DECL FDAT FP589={TOOL_NO 0,BASE_NO 0,IPO_FRAME #BASE,POINT2[] " ",TQ_STATE FALSE}
DECL E6POS XP589={X 12666.37592,Y -538.48386,Z 3708.53974,A -127.07895,B -20.60151,C -3.44033,S 2,T 35,E1 -10812.08896,E2 0,E3 0,E4 0,E5 0,E6 0}
; DECL LDAT LCPDATP113={VEL 1,ACC 100,APO_DIST 100,APO_FAC 50.0,ORI_TYP #VAR,CIRC_TYP #BASE,JERK_FAC 50.0}
DECL FDAT FP590={TOOL_NO 0,BASE_NO 0,IPO_FRAME #BASE,POINT2[] " ",TQ_STATE FALSE}
DECL E6POS XP590={X 6379.94734,Y -681.40788,Z 3158.20554,A -102.40256,B 11.37187,C 4.81103,S 2,T 35,E1 -4209.91162,E2 0,E3 0,E4 0,E5 0,E6 0}
; DECL LDAT LCPDATP114={VEL 1,ACC 100,APO_DIST 100,APO_FAC 50.0,ORI_TYP #VAR,CIRC_TYP #BASE,JERK_FAC 50.0}
DECL FDAT FP591={TOOL_NO 0,BASE_NO 0,IPO_FRAME #BASE,POINT2[] " ",TQ_STATE FALSE}
DECL E6POS XP591={X 6328.481,Y -681.40737,Z 3158.20597,A -102.7078,B 7.77597,C 4.76025,S 2,T 35,E1 -4158.44503,E2 0,E3 0,E4 0,E5 0,E6 0}
; DECL LDAT LCPDATP115={VEL 1,ACC 100,APO_DIST 100,APO_FAC 50.0,ORI_TYP #VAR,CIRC_TYP #BASE,JERK_FAC 50.0}
DECL FDAT FP592={TOOL_NO 0,BASE_NO 0,IPO_FRAME #BASE,POINT2[] " ",TQ_STATE FALSE}
DECL E6POS XP592={X 12929.38089,Y -681.40737,Z 3158.20639,A -83.4604,B -12.81532,C -0.94267,S 2,T 35,E1 -10812.08896,E2 0,E3 0,E4 0,E5 0,E6 0}
; DECL LDAT LCPDATP116={VEL 1,ACC 100,APO_DIST 100,APO_FAC 50.0,ORI_TYP #VAR,CIRC_TYP #BASE,JERK_FAC 50.0}
DECL FDAT FP593={TOOL_NO 0,BASE_NO 0,IPO_FRAME #BASE,POINT2[] " ",TQ_STATE FALSE}
DECL E6POS XP593={X 12886.08572,Y -646.4113,Z 3336.02814,A -83.4604,B -12.81532,C -0.94267,S 2,T 35,E1 -10812.08896,E2 0,E3 0,E4 0,E5 0,E6 0}
; DECL LDAT LCPDATP117={VEL 1,ACC 100,APO_DIST 100,APO_FAC 50.0,ORI_TYP #VAR,CIRC_TYP #BASE,JERK_FAC 50.0}
DECL FDAT FP594={TOOL_NO 0,BASE_NO 0,IPO_FRAME #BASE,POINT2[] " ",TQ_STATE FALSE}
DECL E6POS XP594={X 6226.20694,Y -691.76303,Z 3410.82553,A -102.7078,B 7.77597,C 4.76022,S 2,T 35,E1 -4167.06683,E2 0,E3 0,E4 0,E5 0,E6 0}
; DECL LDAT LCPDATP118={VEL 1,ACC 100,APO_DIST 100,APO_FAC 50.0,ORI_TYP #VAR,CIRC_TYP #BASE,JERK_FAC 50.0}
DECL FDAT FP595={TOOL_NO 0,BASE_NO 0,IPO_FRAME #BASE,POINT2[] " ",TQ_STATE FALSE}
DECL E6POS XP595={X 6109.20944,Y -705.3695,Z 3654.40552,A -102.70779,B 7.77597,C 4.76025,S 2,T 35,E1 -4140.9372,E2 0,E3 0,E4 0,E5 0,E6 0}
; DECL LDAT LCPDATP121={VEL 1,ACC 100,APO_DIST 100,APO_FAC 50.0,ORI_TYP #VAR,CIRC_TYP #BASE,JERK_FAC 50.0}
DECL FDAT FP596={TOOL_NO 0,BASE_NO 0,IPO_FRAME #BASE,POINT2[] " ",TQ_STATE FALSE}
DECL E6POS XP596={X 12777.06723,Y -602.17839,Z 3573.69413,A -83.4604,B -12.81532,C -0.94267,S 2,T 35,E1 -10812.08896,E2 0,E3 0,E4 0,E5 0,E6 0}
; DECL LDAT LCPDATP122={VEL 1,ACC 100,APO_DIST 100,APO_FAC 50.0,ORI_TYP #VAR,CIRC_TYP #BASE,JERK_FAC 50.0}
DECL FDAT FP597={TOOL_NO 0,BASE_NO 0,IPO_FRAME #BASE,POINT2[] " ",TQ_STATE FALSE}
DECL E6POS XP597={X 12675.92788,Y -569.18264,Z 3775.2407,A -83.4604,B -12.81532,C -0.94267,S 2,T 35,E1 -10812.08896,E2 0,E3 0,E4 0,E5 0,E6 0}
; DECL LDAT LCPDATP119={VEL 1,ACC 100,APO_DIST 100,APO_FAC 50.0,ORI_TYP #VAR,CIRC_TYP #BASE,JERK_FAC 50.0}
DECL FDAT FP598={TOOL_NO 0,BASE_NO 0,IPO_FRAME #BASE,POINT2[] " ",TQ_STATE FALSE}
DECL E6POS XP598={X 6034.81499,Y -708.12179,Z 3847.76366,A -102.7078,B 7.77596,C 4.76026,S 2,T 35,E1 -4174.36752,E2 0,E3 0,E4 0,E5 0,E6 0}
; DECL LDAT LCPDATP120={VEL 1,ACC 100,APO_DIST 100,APO_FAC 50.0,ORI_TYP #VAR,CIRC_TYP #BASE,JERK_FAC 50.0}
DECL FDAT FP599={TOOL_NO 0,BASE_NO 0,IPO_FRAME #BASE,POINT2[] " ",TQ_STATE FALSE}
DECL E6POS XP599={X 5808.56571,Y -717.10091,Z 4003.7046,A -102.70779,B 7.77596,C 4.76025,S 2,T 35,E1 -4005.10214,E2 0,E3 0,E4 0,E5 0,E6 0}
; DECL LDAT LCPDATP123={VEL 1,ACC 100,APO_DIST 100,APO_FAC 50.0,ORI_TYP #VAR,CIRC_TYP #BASE,JERK_FAC 50.0}
DECL FDAT FP600={TOOL_NO 0,BASE_NO 0,IPO_FRAME #BASE,POINT2[] " ",TQ_STATE FALSE}
DECL E6POS XP600={X 12607.03936,Y -538.48386,Z 3940.5062,A -83.4604,B -12.81532,C -0.94267,S 2,T 35,E1 -10812.08896,E2 0,E3 0,E4 0,E5 0,E6 0}
; DECL LDAT LCPDATP124={VEL 1,ACC 100,APO_DIST 100,APO_FAC 50.0,ORI_TYP #VAR,CIRC_TYP #BASE,JERK_FAC 50.0}
DECL FDAT FP601={TOOL_NO 0,BASE_NO 0,IPO_FRAME #BASE,POINT2[] " ",TQ_STATE FALSE}
DECL E6POS XP601={X 12329.73693,Y -538.48386,Z 3940.5062,A -83.38777,B -15.32829,C -1.2413,S 2,T 35,E1 -10812.08896,E2 0,E3 0,E4 0,E5 0,E6 0}
; DECL LDAT LCPDATP130={VEL 1,ACC 100,APO_DIST 100,APO_FAC 50.0,ORI_TYP #VAR,CIRC_TYP #BASE,JERK_FAC 50.0}
DECL FDAT FP602={TOOL_NO 0,BASE_NO 0,IPO_FRAME #BASE,POINT2[] " ",TQ_STATE FALSE}
DECL E6POS XP602={X 6035.27715,Y -717.10158,Z 4003.70466,A -106.51042,B 6.34838,C 5.00917,S 2,T 35,E1 -4231.81368,E2 0,E3 0,E4 0,E5 0,E6 0}
; DECL LDAT LCPDATP131={VEL 1,ACC 100,APO_DIST 100,APO_FAC 50.0,ORI_TYP #VAR,CIRC_TYP #BASE,JERK_FAC 50.0}
DECL FDAT FP603={TOOL_NO 0,BASE_NO 0,IPO_FRAME #BASE,POINT2[] " ",TQ_STATE FALSE}
DECL E6POS XP603={X 6001.84737,Y -717.10113,Z 4003.70421,A -106.4599,B 4.5615,C 5.54032,S 2,T 35,E1 -4198.38336,E2 0,E3 0,E4 0,E5 0,E6 0}
; DECL LDAT LCPDATP125={VEL 1,ACC 100,APO_DIST 100,APO_FAC 50.0,ORI_TYP #VAR,CIRC_TYP #BASE,JERK_FAC 50.0}
DECL FDAT FP604={TOOL_NO 0,BASE_NO 0,IPO_FRAME #BASE,POINT2[] " ",TQ_STATE FALSE}
DECL E6POS XP604={X 12327.62864,Y -538.48366,Z 3940.50597,A -87.76623,B -17.49847,C -1.50503,S 2,T 35,E1 -10473.34117,E2 0,E3 0,E4 0,E5 0,E6 0}
; DECL LDAT LCPDATP126={VEL 1,ACC 100,APO_DIST 100,APO_FAC 50.0,ORI_TYP #VAR,CIRC_TYP #BASE,JERK_FAC 50.0}
DECL FDAT FP605={TOOL_NO 0,BASE_NO 0,IPO_FRAME #BASE,POINT2[] " ",TQ_STATE FALSE}
DECL E6POS XP605={X 12344.44126,Y -538.48354,Z 3940.50612,A -92.12133,B -19.55447,C -1.59012,S 2,T 35,E1 -10490.15446,E2 0,E3 0,E4 0,E5 0,E6 0}
; DECL LDAT LCPDATP132={VEL 1,ACC 100,APO_DIST 100,APO_FAC 50.0,ORI_TYP #VAR,CIRC_TYP #BASE,JERK_FAC 50.0}
DECL FDAT FP606={TOOL_NO 0,BASE_NO 0,IPO_FRAME #BASE,POINT2[] " ",TQ_STATE FALSE}
DECL E6POS XP606={X 5984.60315,Y -717.10142,Z 4003.7045,A -107.27293,B 2.66443,C 6.10126,S 2,T 35,E1 -4181.13976,E2 0,E3 0,E4 0,E5 0,E6 0}
; DECL LDAT LCPDATP133={VEL 1,ACC 100,APO_DIST 100,APO_FAC 50.0,ORI_TYP #VAR,CIRC_TYP #BASE,JERK_FAC 50.0}
DECL FDAT FP607={TOOL_NO 0,BASE_NO 0,IPO_FRAME #BASE,POINT2[] " ",TQ_STATE FALSE}
DECL E6POS XP607={X 5959.53065,Y -717.10165,Z 4003.70439,A -107.25516,B 0.74219,C 6.69889,S 2,T 35,E1 -4156.06702,E2 0,E3 0,E4 0,E5 0,E6 0}
; DECL LDAT LCPDATP127={VEL 1,ACC 100,APO_DIST 100,APO_FAC 50.0,ORI_TYP #VAR,CIRC_TYP #BASE,JERK_FAC 50.0}
DECL FDAT FP608={TOOL_NO 0,BASE_NO 0,IPO_FRAME #BASE,POINT2[] " ",TQ_STATE FALSE}
DECL E6POS XP608={X 12327.65948,Y -538.48376,Z 3940.50627,A -96.02004,B -21.56802,C -1.50992,S 2,T 35,E1 -10473.37259,E2 0,E3 0,E4 0,E5 0,E6 0}
; DECL LDAT LCPDATP128={VEL 1,ACC 100,APO_DIST 100,APO_FAC 50.0,ORI_TYP #VAR,CIRC_TYP #BASE,JERK_FAC 50.0}
DECL FDAT FP609={TOOL_NO 0,BASE_NO 0,IPO_FRAME #BASE,POINT2[] " ",TQ_STATE FALSE}
DECL E6POS XP609={X 12434.40962,Y -538.48361,Z 3791.38491,A -100.48203,B -23.59142,C -1.27711,S 2,T 35,E1 -10580.12251,E2 0,E3 0,E4 0,E5 0,E6 0}
; DECL LDAT LCPDATP134={VEL 1,ACC 100,APO_DIST 100,APO_FAC 50.0,ORI_TYP #VAR,CIRC_TYP #BASE,JERK_FAC 50.0}
DECL FDAT FP610={TOOL_NO 0,BASE_NO 0,IPO_FRAME #BASE,POINT2[] " ",TQ_STATE FALSE}
DECL E6POS XP610={X 6027.18413,Y -717.10157,Z 4003.70451,A -108.83879,B -1.2655,C 7.3225,S 2,T 35,E1 -4223.72032,E2 0,E3 0,E4 0,E5 0,E6 0}
; DECL LDAT LCPDATP135={VEL 1,ACC 100,APO_DIST 100,APO_FAC 50.0,ORI_TYP #VAR,CIRC_TYP #BASE,JERK_FAC 50.0}
DECL FDAT FP611={TOOL_NO 0,BASE_NO 0,IPO_FRAME #BASE,POINT2[] " ",TQ_STATE FALSE}
DECL E6POS XP611={X 5994.01853,Y -717.10159,Z 4003.70409,A -109.42003,B -3.44272,C 8.06654,S 2,T 35,E1 -4190.55423,E2 0,E3 0,E4 0,E5 0,E6 0}
; DECL LDAT LCPDATP129={VEL 1,ACC 100,APO_DIST 100,APO_FAC 50.0,ORI_TYP #VAR,CIRC_TYP #BASE,JERK_FAC 50.0}
DECL FDAT FP612={TOOL_NO 0,BASE_NO 0,IPO_FRAME #BASE,POINT2[] " ",TQ_STATE FALSE}
DECL E6POS XP612={X 12525.53957,Y -538.48385,Z 3733.39322,A -103.74147,B -24.12805,C -1.24549,S 2,T 35,E1 -10671.25219,E2 0,E3 0,E4 0,E5 0,E6 0}
; DECL LDAT LCPDATP138={VEL 1,ACC 100,APO_DIST 100,APO_FAC 50.0,ORI_TYP #VAR,CIRC_TYP #BASE,JERK_FAC 50.0}
DECL FDAT FP613={TOOL_NO 0,BASE_NO 0,IPO_FRAME #BASE,POINT2[] " ",TQ_STATE FALSE}
DECL E6POS XP613={X 12409.55634,Y -538.48385,Z 3733.39322,A -103.74147,B -24.12805,C -1.24549,S 2,T 35,E1 -10555.26896,E2 0,E3 0,E4 0,E5 0,E6 0}
; DECL LDAT LCPDATP136={VEL 1,ACC 100,APO_DIST 100,APO_FAC 50.0,ORI_TYP #VAR,CIRC_TYP #BASE,JERK_FAC 50.0}
DECL FDAT FP614={TOOL_NO 0,BASE_NO 0,IPO_FRAME #BASE,POINT2[] " ",TQ_STATE FALSE}
DECL E6POS XP614={X 5960.30101,Y -717.10136,Z 4003.70387,A -109.95564,B -5.51238,C 8.79955,S 2,T 35,E1 -4156.83652,E2 0,E3 0,E4 0,E5 0,E6 0}
; DECL LDAT LCPDATP137={VEL 1,ACC 100,APO_DIST 100,APO_FAC 50.0,ORI_TYP #VAR,CIRC_TYP #BASE,JERK_FAC 50.0}
DECL FDAT FP615={TOOL_NO 0,BASE_NO 0,IPO_FRAME #BASE,POINT2[] " ",TQ_STATE FALSE}
DECL E6POS XP615={X 5959.29294,Y -717.10098,Z 4003.70454,A -110.58224,B -7.77816,C 9.62993,S 2,T 35,E1 -4155.82897,E2 0,E3 0,E4 0,E5 0,E6 0}
; DECL LDAT LCPDATP139={VEL 1,ACC 100,APO_DIST 100,APO_FAC 50.0,ORI_TYP #VAR,CIRC_TYP #BASE,JERK_FAC 50.0}
DECL FDAT FP616={TOOL_NO 0,BASE_NO 0,IPO_FRAME #BASE,POINT2[] " ",TQ_STATE FALSE}
DECL E6POS XP616={X 12666.37592,Y -538.48386,Z 3733.39329,A -110.95703,B -23.34196,C -1.63568,S 2,T 35,E1 -10812.08896,E2 0,E3 0,E4 0,E5 0,E6 0}
; DECL LDAT LCPDATP140={VEL 1,ACC 100,APO_DIST 100,APO_FAC 50.0,ORI_TYP #VAR,CIRC_TYP #BASE,JERK_FAC 50.0}
DECL FDAT FP617={TOOL_NO 0,BASE_NO 0,IPO_FRAME #BASE,POINT2[] " ",TQ_STATE FALSE}
DECL E6POS XP617={X 12666.37592,Y -538.48386,Z 3700.25522,A -113.36831,B -23.34196,C -1.63568,S 2,T 35,E1 -10812.08896,E2 0,E3 0,E4 0,E5 0,E6 0}
; DECL LDAT LCPDATP149={VEL 1,ACC 100,APO_DIST 100,APO_FAC 50.0,ORI_TYP #VAR,CIRC_TYP #BASE,JERK_FAC 50.0}
DECL FDAT FP618={TOOL_NO 0,BASE_NO 0,IPO_FRAME #BASE,POINT2[] " ",TQ_STATE FALSE}
DECL E6POS XP618={X 5916.8006,Y -717.10155,Z 4003.70412,A -110.72224,B -10.13455,C 10.52896,S 2,T 35,E1 -4113.33656,E2 0,E3 0,E4 0,E5 0,E6 0}
; DECL LDAT LCPDATP150={VEL 1,ACC 100,APO_DIST 100,APO_FAC 50.0,ORI_TYP #VAR,CIRC_TYP #BASE,JERK_FAC 50.0}
DECL FDAT FP619={TOOL_NO 0,BASE_NO 0,IPO_FRAME #BASE,POINT2[] " ",TQ_STATE FALSE}
DECL E6POS XP619={X 5875.31565,Y -717.1012,Z 4003.70448,A -110.8879,B -12.32973,C 11.37928,S 2,T 35,E1 -4071.85169,E2 0,E3 0,E4 0,E5 0,E6 0}
; DECL LDAT LCPDATP141={VEL 1,ACC 100,APO_DIST 100,APO_FAC 50.0,ORI_TYP #VAR,CIRC_TYP #BASE,JERK_FAC 50.0}
DECL FDAT FP620={TOOL_NO 0,BASE_NO 0,IPO_FRAME #BASE,POINT2[] " ",TQ_STATE FALSE}
DECL E6POS XP620={X 12666.37592,Y -538.48386,Z 3675.40167,A -115.34787,B -23.34196,C -1.63568,S 2,T 35,E1 -10812.08896,E2 0,E3 0,E4 0,E5 0,E6 0}
; DECL LDAT LCPDATP142={VEL 1,ACC 100,APO_DIST 100,APO_FAC 50.0,ORI_TYP #VAR,CIRC_TYP #BASE,JERK_FAC 50.0}
DECL FDAT FP621={TOOL_NO 0,BASE_NO 0,IPO_FRAME #BASE,POINT2[] " ",TQ_STATE FALSE}
DECL E6POS XP621={X 12666.37592,Y -538.48386,Z 3725.10877,A -117.62399,B -22.31862,C -2.21953,S 2,T 35,E1 -10812.08896,E2 0,E3 0,E4 0,E5 0,E6 0}
; DECL LDAT LCPDATP151={VEL 1,ACC 100,APO_DIST 100,APO_FAC 50.0,ORI_TYP #VAR,CIRC_TYP #BASE,JERK_FAC 50.0}
DECL FDAT FP622={TOOL_NO 0,BASE_NO 0,IPO_FRAME #BASE,POINT2[] " ",TQ_STATE FALSE}
DECL E6POS XP622={X 5898.57722,Y -717.10122,Z 4003.70435,A -112.09203,B -14.38754,C 12.19033,S 2,T 35,E1 -4095.11298,E2 0,E3 0,E4 0,E5 0,E6 0}
; DECL LDAT LCPDATP152={VEL 1,ACC 100,APO_DIST 100,APO_FAC 50.0,ORI_TYP #VAR,CIRC_TYP #BASE,JERK_FAC 50.0}
DECL FDAT FP623={TOOL_NO 0,BASE_NO 0,IPO_FRAME #BASE,POINT2[] " ",TQ_STATE FALSE}
DECL E6POS XP623={X 5854.40488,Y -717.10171,Z 4003.70448,A -112.35649,B -16.71303,C 13.17652,S 2,T 35,E1 -4050.94133,E2 0,E3 0,E4 0,E5 0,E6 0}
; DECL LDAT LCPDATP143={VEL 1,ACC 100,APO_DIST 100,APO_FAC 50.0,ORI_TYP #VAR,CIRC_TYP #BASE,JERK_FAC 50.0}
DECL FDAT FP624={TOOL_NO 0,BASE_NO 0,IPO_FRAME #BASE,POINT2[] " ",TQ_STATE FALSE}
DECL E6POS XP624={X 12666.37592,Y -538.48386,Z 3708.53974,A -119.39266,B -22.0406,C -2.38888,S 2,T 35,E1 -10812.08896,E2 0,E3 0,E4 0,E5 0,E6 0}
; DECL LDAT LCPDATP144={VEL 1,ACC 100,APO_DIST 100,APO_FAC 50.0,ORI_TYP #VAR,CIRC_TYP #BASE,JERK_FAC 50.0}
DECL FDAT FP625={TOOL_NO 0,BASE_NO 0,IPO_FRAME #BASE,POINT2[] " ",TQ_STATE FALSE}
DECL E6POS XP625={X 12666.37592,Y -538.48386,Z 3716.82426,A -121.52366,B -21.70131,C -2.61349,S 2,T 35,E1 -10812.08896,E2 0,E3 0,E4 0,E5 0,E6 0}
; DECL LDAT LCPDATP153={VEL 1,ACC 100,APO_DIST 100,APO_FAC 50.0,ORI_TYP #VAR,CIRC_TYP #BASE,JERK_FAC 50.0}
DECL FDAT FP626={TOOL_NO 0,BASE_NO 0,IPO_FRAME #BASE,POINT2[] " ",TQ_STATE FALSE}
DECL E6POS XP626={X 5865.70091,Y -717.10124,Z 4003.70383,A -113.62634,B -18.80667,C 14.08679,S 2,T 35,E1 -4062.23613,E2 0,E3 0,E4 0,E5 0,E6 0}
; DECL LDAT LCPDATP154={VEL 1,ACC 100,APO_DIST 100,APO_FAC 50.0,ORI_TYP #VAR,CIRC_TYP #BASE,JERK_FAC 50.0}
DECL FDAT FP627={TOOL_NO 0,BASE_NO 0,IPO_FRAME #BASE,POINT2[] " ",TQ_STATE FALSE}
DECL E6POS XP627={X 5786.97193,Y -717.10138,Z 4003.70442,A -113.90846,B -20.59534,C 14.92344,S 2,T 35,E1 -3983.50839,E2 0,E3 0,E4 0,E5 0,E6 0}
; DECL LDAT LCPDATP145={VEL 1,ACC 100,APO_DIST 100,APO_FAC 50.0,ORI_TYP #VAR,CIRC_TYP #BASE,JERK_FAC 50.0}
DECL FDAT FP628={TOOL_NO 0,BASE_NO 0,IPO_FRAME #BASE,POINT2[] " ",TQ_STATE FALSE}
DECL E6POS XP628={X 12666.37592,Y -538.48386,Z 3691.97071,A -122.58569,B -21.70131,C -2.61349,S 2,T 35,E1 -10812.08896,E2 0,E3 0,E4 0,E5 0,E6 0}
; DECL LDAT LCPDATP146={VEL 1,ACC 100,APO_DIST 100,APO_FAC 50.0,ORI_TYP #VAR,CIRC_TYP #BASE,JERK_FAC 50.0}
DECL FDAT FP629={TOOL_NO 0,BASE_NO 0,IPO_FRAME #BASE,POINT2[] " ",TQ_STATE FALSE}
DECL E6POS XP629={X 12666.37592,Y -538.48386,Z 3741.67781,A -124.88801,B -20.60151,C -3.44033,S 2,T 35,E1 -10812.08896,E2 0,E3 0,E4 0,E5 0,E6 0}
; DECL LDAT LCPDATP155={VEL 1,ACC 100,APO_DIST 100,APO_FAC 50.0,ORI_TYP #VAR,CIRC_TYP #BASE,JERK_FAC 50.0}
DECL FDAT FP630={TOOL_NO 0,BASE_NO 0,IPO_FRAME #BASE,POINT2[] " ",TQ_STATE FALSE}
DECL E6POS XP630={X 5766.06143,Y -717.10078,Z 4003.7047,A -114.88478,B -21.82725,C 15.51221,S 2,T 35,E1 -3962.59803,E2 0,E3 0,E4 0,E5 0,E6 0}
; DECL LDAT LCPDATP156={VEL 1,ACC 100,APO_DIST 100,APO_FAC 50.0,ORI_TYP #VAR,CIRC_TYP #BASE,JERK_FAC 50.0}
DECL FDAT FP631={TOOL_NO 0,BASE_NO 0,IPO_FRAME #BASE,POINT2[] " ",TQ_STATE FALSE}
DECL E6POS XP631={X 5671.46198,Y -717.1018,Z 4003.704,A -116.65787,B -23.21109,C 16.21129,S 2,T 35,E1 -3867.99764,E2 0,E3 0,E4 0,E5 0,E6 0}
; DECL LDAT LCPDATP147={VEL 1,ACC 100,APO_DIST 100,APO_FAC 50.0,ORI_TYP #VAR,CIRC_TYP #BASE,JERK_FAC 50.0}
DECL FDAT FP632={TOOL_NO 0,BASE_NO 0,IPO_FRAME #BASE,POINT2[] " ",TQ_STATE FALSE}
DECL E6POS XP632={X 12666.37592,Y -538.48386,Z 3708.53974,A -127.07895,B -20.60151,C -3.44033,S 2,T 35,E1 -10812.08896,E2 0,E3 0,E4 0,E5 0,E6 0}
; DECL LDAT LCPDATP113={VEL 1,ACC 100,APO_DIST 100,APO_FAC 50.0,ORI_TYP #VAR,CIRC_TYP #BASE,JERK_FAC 50.0}
DECL FDAT FP633={TOOL_NO 0,BASE_NO 0,IPO_FRAME #BASE,POINT2[] " ",TQ_STATE FALSE}
DECL E6POS XP633={X 6379.94734,Y -681.40788,Z 3158.20554,A -102.40256,B 11.37187,C 4.81103,S 2,T 35,E1 -4209.91162,E2 0,E3 0,E4 0,E5 0,E6 0}
; DECL LDAT LCPDATP114={VEL 1,ACC 100,APO_DIST 100,APO_FAC 50.0,ORI_TYP #VAR,CIRC_TYP #BASE,JERK_FAC 50.0}
DECL FDAT FP634={TOOL_NO 0,BASE_NO 0,IPO_FRAME #BASE,POINT2[] " ",TQ_STATE FALSE}
DECL E6POS XP634={X 6328.481,Y -681.40737,Z 3158.20597,A -102.7078,B 7.77597,C 4.76025,S 2,T 35,E1 -4158.44503,E2 0,E3 0,E4 0,E5 0,E6 0}
; DECL LDAT LCPDATP115={VEL 1,ACC 100,APO_DIST 100,APO_FAC 50.0,ORI_TYP #VAR,CIRC_TYP #BASE,JERK_FAC 50.0}
DECL FDAT FP635={TOOL_NO 0,BASE_NO 0,IPO_FRAME #BASE,POINT2[] " ",TQ_STATE FALSE}
DECL E6POS XP635={X 12929.38089,Y -681.40737,Z 3158.20639,A -83.4604,B -12.81532,C -0.94267,S 2,T 35,E1 -10812.08896,E2 0,E3 0,E4 0,E5 0,E6 0}
; DECL LDAT LCPDATP116={VEL 1,ACC 100,APO_DIST 100,APO_FAC 50.0,ORI_TYP #VAR,CIRC_TYP #BASE,JERK_FAC 50.0}
DECL FDAT FP636={TOOL_NO 0,BASE_NO 0,IPO_FRAME #BASE,POINT2[] " ",TQ_STATE FALSE}
DECL E6POS XP636={X 12886.08572,Y -646.4113,Z 3336.02814,A -83.4604,B -12.81532,C -0.94267,S 2,T 35,E1 -10812.08896,E2 0,E3 0,E4 0,E5 0,E6 0}
; DECL LDAT LCPDATP117={VEL 1,ACC 100,APO_DIST 100,APO_FAC 50.0,ORI_TYP #VAR,CIRC_TYP #BASE,JERK_FAC 50.0}
DECL FDAT FP637={TOOL_NO 0,BASE_NO 0,IPO_FRAME #BASE,POINT2[] " ",TQ_STATE FALSE}
DECL E6POS XP637={X 6226.20694,Y -691.76303,Z 3410.82553,A -102.7078,B 7.77597,C 4.76022,S 2,T 35,E1 -4167.06683,E2 0,E3 0,E4 0,E5 0,E6 0}
; DECL LDAT LCPDATP118={VEL 1,ACC 100,APO_DIST 100,APO_FAC 50.0,ORI_TYP #VAR,CIRC_TYP #BASE,JERK_FAC 50.0}
DECL FDAT FP638={TOOL_NO 0,BASE_NO 0,IPO_FRAME #BASE,POINT2[] " ",TQ_STATE FALSE}
DECL E6POS XP638={X 6109.20944,Y -705.3695,Z 3654.40552,A -102.70779,B 7.77597,C 4.76025,S 2,T 35,E1 -4140.9372,E2 0,E3 0,E4 0,E5 0,E6 0}
; DECL LDAT LCPDATP121={VEL 1,ACC 100,APO_DIST 100,APO_FAC 50.0,ORI_TYP #VAR,CIRC_TYP #BASE,JERK_FAC 50.0}
DECL FDAT FP639={TOOL_NO 0,BASE_NO 0,IPO_FRAME #BASE,POINT2[] " ",TQ_STATE FALSE}
DECL E6POS XP639={X 12777.06723,Y -602.17839,Z 3573.69413,A -83.4604,B -12.81532,C -0.94267,S 2,T 35,E1 -10812.08896,E2 0,E3 0,E4 0,E5 0,E6 0}
; DECL LDAT LCPDATP122={VEL 1,ACC 100,APO_DIST 100,APO_FAC 50.0,ORI_TYP #VAR,CIRC_TYP #BASE,JERK_FAC 50.0}
DECL FDAT FP640={TOOL_NO 0,BASE_NO 0,IPO_FRAME #BASE,POINT2[] " ",TQ_STATE FALSE}
DECL E6POS XP640={X 12675.92788,Y -569.18264,Z 3775.2407,A -83.4604,B -12.81532,C -0.94267,S 2,T 35,E1 -10812.08896,E2 0,E3 0,E4 0,E5 0,E6 0}
; DECL LDAT LCPDATP119={VEL 1,ACC 100,APO_DIST 100,APO_FAC 50.0,ORI_TYP #VAR,CIRC_TYP #BASE,JERK_FAC 50.0}
DECL FDAT FP641={TOOL_NO 0,BASE_NO 0,IPO_FRAME #BASE,POINT2[] " ",TQ_STATE FALSE}
DECL E6POS XP641={X 6034.81499,Y -708.12179,Z 3847.76366,A -102.7078,B 7.77596,C 4.76026,S 2,T 35,E1 -4174.36752,E2 0,E3 0,E4 0,E5 0,E6 0}
; DECL LDAT LCPDATP120={VEL 1,ACC 100,APO_DIST 100,APO_FAC 50.0,ORI_TYP #VAR,CIRC_TYP #BASE,JERK_FAC 50.0}
DECL FDAT FP642={TOOL_NO 0,BASE_NO 0,IPO_FRAME #BASE,POINT2[] " ",TQ_STATE FALSE}
DECL E6POS XP642={X 5808.56571,Y -717.10091,Z 4003.7046,A -102.70779,B 7.77596,C 4.76025,S 2,T 35,E1 -4005.10214,E2 0,E3 0,E4 0,E5 0,E6 0}
; DECL LDAT LCPDATP123={VEL 1,ACC 100,APO_DIST 100,APO_FAC 50.0,ORI_TYP #VAR,CIRC_TYP #BASE,JERK_FAC 50.0}
DECL FDAT FP643={TOOL_NO 0,BASE_NO 0,IPO_FRAME #BASE,POINT2[] " ",TQ_STATE FALSE}
DECL E6POS XP643={X 12607.03936,Y -538.48386,Z 3940.5062,A -83.4604,B -12.81532,C -0.94267,S 2,T 35,E1 -10812.08896,E2 0,E3 0,E4 0,E5 0,E6 0}
; DECL LDAT LCPDATP124={VEL 1,ACC 100,APO_DIST 100,APO_FAC 50.0,ORI_TYP #VAR,CIRC_TYP #BASE,JERK_FAC 50.0}
DECL FDAT FP644={TOOL_NO 0,BASE_NO 0,IPO_FRAME #BASE,POINT2[] " ",TQ_STATE FALSE}
DECL E6POS XP644={X 12329.73693,Y -538.48386,Z 3940.5062,A -83.38777,B -15.32829,C -1.2413,S 2,T 35,E1 -10812.08896,E2 0,E3 0,E4 0,E5 0,E6 0}
; DECL LDAT LCPDATP130={VEL 1,ACC 100,APO_DIST 100,APO_FAC 50.0,ORI_TYP #VAR,CIRC_TYP #BASE,JERK_FAC 50.0}
DECL FDAT FP645={TOOL_NO 0,BASE_NO 0,IPO_FRAME #BASE,POINT2[] " ",TQ_STATE FALSE}
DECL E6POS XP645={X 6035.27715,Y -717.10158,Z 4003.70466,A -106.51042,B 6.34838,C 5.00917,S 2,T 35,E1 -4231.81368,E2 0,E3 0,E4 0,E5 0,E6 0}
; DECL LDAT LCPDATP131={VEL 1,ACC 100,APO_DIST 100,APO_FAC 50.0,ORI_TYP #VAR,CIRC_TYP #BASE,JERK_FAC 50.0}
DECL FDAT FP646={TOOL_NO 0,BASE_NO 0,IPO_FRAME #BASE,POINT2[] " ",TQ_STATE FALSE}
DECL E6POS XP646={X 6001.84737,Y -717.10113,Z 4003.70421,A -106.4599,B 4.5615,C 5.54032,S 2,T 35,E1 -4198.38336,E2 0,E3 0,E4 0,E5 0,E6 0}
; DECL LDAT LCPDATP125={VEL 1,ACC 100,APO_DIST 100,APO_FAC 50.0,ORI_TYP #VAR,CIRC_TYP #BASE,JERK_FAC 50.0}
DECL FDAT FP647={TOOL_NO 0,BASE_NO 0,IPO_FRAME #BASE,POINT2[] " ",TQ_STATE FALSE}
DECL E6POS XP647={X 12327.62864,Y -538.48366,Z 3940.50597,A -87.76623,B -17.49847,C -1.50503,S 2,T 35,E1 -10473.34117,E2 0,E3 0,E4 0,E5 0,E6 0}
; DECL LDAT LCPDATP126={VEL 1,ACC 100,APO_DIST 100,APO_FAC 50.0,ORI_TYP #VAR,CIRC_TYP #BASE,JERK_FAC 50.0}
DECL FDAT FP648={TOOL_NO 0,BASE_NO 0,IPO_FRAME #BASE,POINT2[] " ",TQ_STATE FALSE}
DECL E6POS XP648={X 12344.44126,Y -538.48354,Z 3940.50612,A -92.12133,B -19.55447,C -1.59012,S 2,T 35,E1 -10490.15446,E2 0,E3 0,E4 0,E5 0,E6 0}
; DECL LDAT LCPDATP132={VEL 1,ACC 100,APO_DIST 100,APO_FAC 50.0,ORI_TYP #VAR,CIRC_TYP #BASE,JERK_FAC 50.0}
DECL FDAT FP649={TOOL_NO 0,BASE_NO 0,IPO_FRAME #BASE,POINT2[] " ",TQ_STATE FALSE}
DECL E6POS XP649={X 5984.60315,Y -717.10142,Z 4003.7045,A -107.27293,B 2.66443,C 6.10126,S 2,T 35,E1 -4181.13976,E2 0,E3 0,E4 0,E5 0,E6 0}
; DECL LDAT LCPDATP133={VEL 1,ACC 100,APO_DIST 100,APO_FAC 50.0,ORI_TYP #VAR,CIRC_TYP #BASE,JERK_FAC 50.0}
DECL FDAT FP650={TOOL_NO 0,BASE_NO 0,IPO_FRAME #BASE,POINT2[] " ",TQ_STATE FALSE}
DECL E6POS XP650={X 5959.53065,Y -717.10165,Z 4003.70439,A -107.25516,B 0.74219,C 6.69889,S 2,T 35,E1 -4156.06702,E2 0,E3 0,E4 0,E5 0,E6 0}
; DECL LDAT LCPDATP127={VEL 1,ACC 100,APO_DIST 100,APO_FAC 50.0,ORI_TYP #VAR,CIRC_TYP #BASE,JERK_FAC 50.0}
DECL FDAT FP651={TOOL_NO 0,BASE_NO 0,IPO_FRAME #BASE,POINT2[] " ",TQ_STATE FALSE}
DECL E6POS XP651={X 12327.65948,Y -538.48376,Z 3940.50627,A -96.02004,B -21.56802,C -1.50992,S 2,T 35,E1 -10473.37259,E2 0,E3 0,E4 0,E5 0,E6 0}
; DECL LDAT LCPDATP128={VEL 1,ACC 100,APO_DIST 100,APO_FAC 50.0,ORI_TYP #VAR,CIRC_TYP #BASE,JERK_FAC 50.0}
DECL FDAT FP652={TOOL_NO 0,BASE_NO 0,IPO_FRAME #BASE,POINT2[] " ",TQ_STATE FALSE}
DECL E6POS XP652={X 12434.40962,Y -538.48361,Z 3791.38491,A -100.48203,B -23.59142,C -1.27711,S 2,T 35,E1 -10580.12251,E2 0,E3 0,E4 0,E5 0,E6 0}
; DECL LDAT LCPDATP134={VEL 1,ACC 100,APO_DIST 100,APO_FAC 50.0,ORI_TYP #VAR,CIRC_TYP #BASE,JERK_FAC 50.0}
DECL FDAT FP653={TOOL_NO 0,BASE_NO 0,IPO_FRAME #BASE,POINT2[] " ",TQ_STATE FALSE}
DECL E6POS XP653={X 6027.18413,Y -717.10157,Z 4003.70451,A -108.83879,B -1.2655,C 7.3225,S 2,T 35,E1 -4223.72032,E2 0,E3 0,E4 0,E5 0,E6 0}
; DECL LDAT LCPDATP135={VEL 1,ACC 100,APO_DIST 100,APO_FAC 50.0,ORI_TYP #VAR,CIRC_TYP #BASE,JERK_FAC 50.0}
DECL FDAT FP654={TOOL_NO 0,BASE_NO 0,IPO_FRAME #BASE,POINT2[] " ",TQ_STATE FALSE}
DECL E6POS XP654={X 5994.01853,Y -717.10159,Z 4003.70409,A -109.42003,B -3.44272,C 8.06654,S 2,T 35,E1 -4190.55423,E2 0,E3 0,E4 0,E5 0,E6 0}
; DECL LDAT LCPDATP129={VEL 1,ACC 100,APO_DIST 100,APO_FAC 50.0,ORI_TYP #VAR,CIRC_TYP #BASE,JERK_FAC 50.0}
DECL FDAT FP655={TOOL_NO 0,BASE_NO 0,IPO_FRAME #BASE,POINT2[] " ",TQ_STATE FALSE}
DECL E6POS XP655={X 12525.53957,Y -538.48385,Z 3733.39322,A -103.74147,B -24.12805,C -1.24549,S 2,T 35,E1 -10671.25219,E2 0,E3 0,E4 0,E5 0,E6 0}
; DECL LDAT LCPDATP138={VEL 1,ACC 100,APO_DIST 100,APO_FAC 50.0,ORI_TYP #VAR,CIRC_TYP #BASE,JERK_FAC 50.0}
DECL FDAT FP656={TOOL_NO 0,BASE_NO 0,IPO_FRAME #BASE,POINT2[] " ",TQ_STATE FALSE}
DECL E6POS XP656={X 12409.55634,Y -538.48385,Z 3733.39322,A -103.74147,B -24.12805,C -1.24549,S 2,T 35,E1 -10555.26896,E2 0,E3 0,E4 0,E5 0,E6 0}
; DECL LDAT LCPDATP136={VEL 1,ACC 100,APO_DIST 100,APO_FAC 50.0,ORI_TYP #VAR,CIRC_TYP #BASE,JERK_FAC 50.0}
DECL FDAT FP657={TOOL_NO 0,BASE_NO 0,IPO_FRAME #BASE,POINT2[] " ",TQ_STATE FALSE}
DECL E6POS XP657={X 5960.30101,Y -717.10136,Z 4003.70387,A -109.95564,B -5.51238,C 8.79955,S 2,T 35,E1 -4156.83652,E2 0,E3 0,E4 0,E5 0,E6 0}
; DECL LDAT LCPDATP137={VEL 1,ACC 100,APO_DIST 100,APO_FAC 50.0,ORI_TYP #VAR,CIRC_TYP #BASE,JERK_FAC 50.0}
DECL FDAT FP658={TOOL_NO 0,BASE_NO 0,IPO_FRAME #BASE,POINT2[] " ",TQ_STATE FALSE}
DECL E6POS XP658={X 5959.29294,Y -717.10098,Z 4003.70454,A -110.58224,B -7.77816,C 9.62993,S 2,T 35,E1 -4155.82897,E2 0,E3 0,E4 0,E5 0,E6 0}
; DECL LDAT LCPDATP139={VEL 1,ACC 100,APO_DIST 100,APO_FAC 50.0,ORI_TYP #VAR,CIRC_TYP #BASE,JERK_FAC 50.0}
DECL FDAT FP659={TOOL_NO 0,BASE_NO 0,IPO_FRAME #BASE,POINT2[] " ",TQ_STATE FALSE}
DECL E6POS XP659={X 12666.37592,Y -538.48386,Z 3733.39329,A -110.95703,B -23.34196,C -1.63568,S 2,T 35,E1 -10812.08896,E2 0,E3 0,E4 0,E5 0,E6 0}
; DECL LDAT LCPDATP140={VEL 1,ACC 100,APO_DIST 100,APO_FAC 50.0,ORI_TYP #VAR,CIRC_TYP #BASE,JERK_FAC 50.0}
DECL FDAT FP660={TOOL_NO 0,BASE_NO 0,IPO_FRAME #BASE,POINT2[] " ",TQ_STATE FALSE}
DECL E6POS XP660={X 12666.37592,Y -538.48386,Z 3700.25522,A -113.36831,B -23.34196,C -1.63568,S 2,T 35,E1 -10812.08896,E2 0,E3 0,E4 0,E5 0,E6 0}
; DECL LDAT LCPDATP149={VEL 1,ACC 100,APO_DIST 100,APO_FAC 50.0,ORI_TYP #VAR,CIRC_TYP #BASE,JERK_FAC 50.0}
DECL FDAT FP661={TOOL_NO 0,BASE_NO 0,IPO_FRAME #BASE,POINT2[] " ",TQ_STATE FALSE}
DECL E6POS XP661={X 5916.8006,Y -717.10155,Z 4003.70412,A -110.72224,B -10.13455,C 10.52896,S 2,T 35,E1 -4113.33656,E2 0,E3 0,E4 0,E5 0,E6 0}
; DECL LDAT LCPDATP150={VEL 1,ACC 100,APO_DIST 100,APO_FAC 50.0,ORI_TYP #VAR,CIRC_TYP #BASE,JERK_FAC 50.0}
DECL FDAT FP662={TOOL_NO 0,BASE_NO 0,IPO_FRAME #BASE,POINT2[] " ",TQ_STATE FALSE}
DECL E6POS XP662={X 5875.31565,Y -717.1012,Z 4003.70448,A -110.8879,B -12.32973,C 11.37928,S 2,T 35,E1 -4071.85169,E2 0,E3 0,E4 0,E5 0,E6 0}
; DECL LDAT LCPDATP141={VEL 1,ACC 100,APO_DIST 100,APO_FAC 50.0,ORI_TYP #VAR,CIRC_TYP #BASE,JERK_FAC 50.0}
DECL FDAT FP663={TOOL_NO 0,BASE_NO 0,IPO_FRAME #BASE,POINT2[] " ",TQ_STATE FALSE}
DECL E6POS XP663={X 12666.37592,Y -538.48386,Z 3675.40167,A -115.34787,B -23.34196,C -1.63568,S 2,T 35,E1 -10812.08896,E2 0,E3 0,E4 0,E5 0,E6 0}
; DECL LDAT LCPDATP142={VEL 1,ACC 100,APO_DIST 100,APO_FAC 50.0,ORI_TYP #VAR,CIRC_TYP #BASE,JERK_FAC 50.0}
DECL FDAT FP664={TOOL_NO 0,BASE_NO 0,IPO_FRAME #BASE,POINT2[] " ",TQ_STATE FALSE}
DECL E6POS XP664={X 12666.37592,Y -538.48386,Z 3725.10877,A -117.62399,B -22.31862,C -2.21953,S 2,T 35,E1 -10812.08896,E2 0,E3 0,E4 0,E5 0,E6 0}
; DECL LDAT LCPDATP151={VEL 1,ACC 100,APO_DIST 100,APO_FAC 50.0,ORI_TYP #VAR,CIRC_TYP #BASE,JERK_FAC 50.0}
DECL FDAT FP665={TOOL_NO 0,BASE_NO 0,IPO_FRAME #BASE,POINT2[] " ",TQ_STATE FALSE}
DECL E6POS XP665={X 5898.57722,Y -717.10122,Z 4003.70435,A -112.09203,B -14.38754,C 12.19033,S 2,T 35,E1 -4095.11298,E2 0,E3 0,E4 0,E5 0,E6 0}
; DECL LDAT LCPDATP152={VEL 1,ACC 100,APO_DIST 100,APO_FAC 50.0,ORI_TYP #VAR,CIRC_TYP #BASE,JERK_FAC 50.0}
DECL FDAT FP666={TOOL_NO 0,BASE_NO 0,IPO_FRAME #BASE,POINT2[] " ",TQ_STATE FALSE}
DECL E6POS XP666={X 5854.40488,Y -717.10171,Z 4003.70448,A -112.35649,B -16.71303,C 13.17652,S 2,T 35,E1 -4050.94133,E2 0,E3 0,E4 0,E5 0,E6 0}
; DECL LDAT LCPDATP143={VEL 1,ACC 100,APO_DIST 100,APO_FAC 50.0,ORI_TYP #VAR,CIRC_TYP #BASE,JERK_FAC 50.0}
DECL FDAT FP667={TOOL_NO 0,BASE_NO 0,IPO_FRAME #BASE,POINT2[] " ",TQ_STATE FALSE}
DECL E6POS XP667={X 12666.37592,Y -538.48386,Z 3708.53974,A -119.39266,B -22.0406,C -2.38888,S 2,T 35,E1 -10812.08896,E2 0,E3 0,E4 0,E5 0,E6 0}
; DECL LDAT LCPDATP144={VEL 1,ACC 100,APO_DIST 100,APO_FAC 50.0,ORI_TYP #VAR,CIRC_TYP #BASE,JERK_FAC 50.0}
DECL FDAT FP668={TOOL_NO 0,BASE_NO 0,IPO_FRAME #BASE,POINT2[] " ",TQ_STATE FALSE}
DECL E6POS XP668={X 12666.37592,Y -538.48386,Z 3716.82426,A -121.52366,B -21.70131,C -2.61349,S 2,T 35,E1 -10812.08896,E2 0,E3 0,E4 0,E5 0,E6 0}
; DECL LDAT LCPDATP153={VEL 1,ACC 100,APO_DIST 100,APO_FAC 50.0,ORI_TYP #VAR,CIRC_TYP #BASE,JERK_FAC 50.0}
DECL FDAT FP669={TOOL_NO 0,BASE_NO 0,IPO_FRAME #BASE,POINT2[] " ",TQ_STATE FALSE}
DECL E6POS XP669={X 5865.70091,Y -717.10124,Z 4003.70383,A -113.62634,B -18.80667,C 14.08679,S 2,T 35,E1 -4062.23613,E2 0,E3 0,E4 0,E5 0,E6 0}
; DECL LDAT LCPDATP154={VEL 1,ACC 100,APO_DIST 100,APO_FAC 50.0,ORI_TYP #VAR,CIRC_TYP #BASE,JERK_FAC 50.0}
DECL FDAT FP670={TOOL_NO 0,BASE_NO 0,IPO_FRAME #BASE,POINT2[] " ",TQ_STATE FALSE}
DECL E6POS XP670={X 5786.97193,Y -717.10138,Z 4003.70442,A -113.90846,B -20.59534,C 14.92344,S 2,T 35,E1 -3983.50839,E2 0,E3 0,E4 0,E5 0,E6 0}
; DECL LDAT LCPDATP145={VEL 1,ACC 100,APO_DIST 100,APO_FAC 50.0,ORI_TYP #VAR,CIRC_TYP #BASE,JERK_FAC 50.0}
DECL FDAT FP671={TOOL_NO 0,BASE_NO 0,IPO_FRAME #BASE,POINT2[] " ",TQ_STATE FALSE}
DECL E6POS XP671={X 12666.37592,Y -538.48386,Z 3691.97071,A -122.58569,B -21.70131,C -2.61349,S 2,T 35,E1 -10812.08896,E2 0,E3 0,E4 0,E5 0,E6 0}
; DECL LDAT LCPDATP146={VEL 1,ACC 100,APO_DIST 100,APO_FAC 50.0,ORI_TYP #VAR,CIRC_TYP #BASE,JERK_FAC 50.0}
DECL FDAT FP672={TOOL_NO 0,BASE_NO 0,IPO_FRAME #BASE,POINT2[] " ",TQ_STATE FALSE}
DECL E6POS XP672={X 12666.37592,Y -538.48386,Z 3741.67781,A -124.88801,B -20.60151,C -3.44033,S 2,T 35,E1 -10812.08896,E2 0,E3 0,E4 0,E5 0,E6 0}
; DECL LDAT LCPDATP155={VEL 1,ACC 100,APO_DIST 100,APO_FAC 50.0,ORI_TYP #VAR,CIRC_TYP #BASE,JERK_FAC 50.0}
DECL FDAT FP673={TOOL_NO 0,BASE_NO 0,IPO_FRAME #BASE,POINT2[] " ",TQ_STATE FALSE}
DECL E6POS XP673={X 5766.06143,Y -717.10078,Z 4003.7047,A -114.88478,B -21.82725,C 15.51221,S 2,T 35,E1 -3962.59803,E2 0,E3 0,E4 0,E5 0,E6 0}
; DECL LDAT LCPDATP156={VEL 1,ACC 100,APO_DIST 100,APO_FAC 50.0,ORI_TYP #VAR,CIRC_TYP #BASE,JERK_FAC 50.0}
DECL FDAT FP674={TOOL_NO 0,BASE_NO 0,IPO_FRAME #BASE,POINT2[] " ",TQ_STATE FALSE}
DECL E6POS XP674={X 5671.46198,Y -717.1018,Z 4003.704,A -116.65787,B -23.21109,C 16.21129,S 2,T 35,E1 -3867.99764,E2 0,E3 0,E4 0,E5 0,E6 0}
; DECL LDAT LCPDATP147={VEL 1,ACC 100,APO_DIST 100,APO_FAC 50.0,ORI_TYP #VAR,CIRC_TYP #BASE,JERK_FAC 50.0}
DECL FDAT FP675={TOOL_NO 0,BASE_NO 0,IPO_FRAME #BASE,POINT2[] " ",TQ_STATE FALSE}
DECL E6POS XP675={X 12666.37592,Y -538.48386,Z 3708.53974,A -127.07895,B -20.60151,C -3.44033,S 2,T 35,E1 -10812.08896,E2 0,E3 0,E4 0,E5 0,E6 0}
; DECL LDAT LCPDATP113={VEL 1,ACC 100,APO_DIST 100,APO_FAC 50.0,ORI_TYP #VAR,CIRC_TYP #BASE,JERK_FAC 50.0}
DECL FDAT FP676={TOOL_NO 0,BASE_NO 0,IPO_FRAME #BASE,POINT2[] " ",TQ_STATE FALSE}
DECL E6POS XP676={X 6379.94734,Y -681.40788,Z 3158.20554,A -102.40256,B 11.37187,C 4.81103,S 2,T 35,E1 -4209.91162,E2 0,E3 0,E4 0,E5 0,E6 0}
; DECL LDAT LCPDATP114={VEL 1,ACC 100,APO_DIST 100,APO_FAC 50.0,ORI_TYP #VAR,CIRC_TYP #BASE,JERK_FAC 50.0}
DECL FDAT FP677={TOOL_NO 0,BASE_NO 0,IPO_FRAME #BASE,POINT2[] " ",TQ_STATE FALSE}
DECL E6POS XP677={X 6328.481,Y -681.40737,Z 3158.20597,A -102.7078,B 7.77597,C 4.76025,S 2,T 35,E1 -4158.44503,E2 0,E3 0,E4 0,E5 0,E6 0}
; DECL LDAT LCPDATP115={VEL 1,ACC 100,APO_DIST 100,APO_FAC 50.0,ORI_TYP #VAR,CIRC_TYP #BASE,JERK_FAC 50.0}
DECL FDAT FP678={TOOL_NO 0,BASE_NO 0,IPO_FRAME #BASE,POINT2[] " ",TQ_STATE FALSE}
DECL E6POS XP678={X 12929.38089,Y -681.40737,Z 3158.20639,A -83.4604,B -12.81532,C -0.94267,S 2,T 35,E1 -10812.08896,E2 0,E3 0,E4 0,E5 0,E6 0}
; DECL LDAT LCPDATP116={VEL 1,ACC 100,APO_DIST 100,APO_FAC 50.0,ORI_TYP #VAR,CIRC_TYP #BASE,JERK_FAC 50.0}
DECL FDAT FP679={TOOL_NO 0,BASE_NO 0,IPO_FRAME #BASE,POINT2[] " ",TQ_STATE FALSE}
DECL E6POS XP679={X 12886.08572,Y -646.4113,Z 3336.02814,A -83.4604,B -12.81532,C -0.94267,S 2,T 35,E1 -10812.08896,E2 0,E3 0,E4 0,E5 0,E6 0}
; DECL LDAT LCPDATP117={VEL 1,ACC 100,APO_DIST 100,APO_FAC 50.0,ORI_TYP #VAR,CIRC_TYP #BASE,JERK_FAC 50.0}
DECL FDAT FP680={TOOL_NO 0,BASE_NO 0,IPO_FRAME #BASE,POINT2[] " ",TQ_STATE FALSE}
DECL E6POS XP680={X 6226.20694,Y -691.76303,Z 3410.82553,A -102.7078,B 7.77597,C 4.76022,S 2,T 35,E1 -4167.06683,E2 0,E3 0,E4 0,E5 0,E6 0}
; DECL LDAT LCPDATP118={VEL 1,ACC 100,APO_DIST 100,APO_FAC 50.0,ORI_TYP #VAR,CIRC_TYP #BASE,JERK_FAC 50.0}
DECL FDAT FP681={TOOL_NO 0,BASE_NO 0,IPO_FRAME #BASE,POINT2[] " ",TQ_STATE FALSE}
DECL E6POS XP681={X 6109.20944,Y -705.3695,Z 3654.40552,A -102.70779,B 7.77597,C 4.76025,S 2,T 35,E1 -4140.9372,E2 0,E3 0,E4 0,E5 0,E6 0}
; DECL LDAT LCPDATP121={VEL 1,ACC 100,APO_DIST 100,APO_FAC 50.0,ORI_TYP #VAR,CIRC_TYP #BASE,JERK_FAC 50.0}
DECL FDAT FP682={TOOL_NO 0,BASE_NO 0,IPO_FRAME #BASE,POINT2[] " ",TQ_STATE FALSE}
DECL E6POS XP682={X 12777.06723,Y -602.17839,Z 3573.69413,A -83.4604,B -12.81532,C -0.94267,S 2,T 35,E1 -10812.08896,E2 0,E3 0,E4 0,E5 0,E6 0}
; DECL LDAT LCPDATP122={VEL 1,ACC 100,APO_DIST 100,APO_FAC 50.0,ORI_TYP #VAR,CIRC_TYP #BASE,JERK_FAC 50.0}
DECL FDAT FP683={TOOL_NO 0,BASE_NO 0,IPO_FRAME #BASE,POINT2[] " ",TQ_STATE FALSE}
DECL E6POS XP683={X 12675.92788,Y -569.18264,Z 3775.2407,A -83.4604,B -12.81532,C -0.94267,S 2,T 35,E1 -10812.08896,E2 0,E3 0,E4 0,E5 0,E6 0}
; DECL LDAT LCPDATP119={VEL 1,ACC 100,APO_DIST 100,APO_FAC 50.0,ORI_TYP #VAR,CIRC_TYP #BASE,JERK_FAC 50.0}
DECL FDAT FP684={TOOL_NO 0,BASE_NO 0,IPO_FRAME #BASE,POINT2[] " ",TQ_STATE FALSE}
DECL E6POS XP684={X 6034.81499,Y -708.12179,Z 3847.76366,A -102.7078,B 7.77596,C 4.76026,S 2,T 35,E1 -4174.36752,E2 0,E3 0,E4 0,E5 0,E6 0}
; DECL LDAT LCPDATP120={VEL 1,ACC 100,APO_DIST 100,APO_FAC 50.0,ORI_TYP #VAR,CIRC_TYP #BASE,JERK_FAC 50.0}
DECL FDAT FP685={TOOL_NO 0,BASE_NO 0,IPO_FRAME #BASE,POINT2[] " ",TQ_STATE FALSE}
DECL E6POS XP685={X 5808.56571,Y -717.10091,Z 4003.7046,A -102.70779,B 7.77596,C 4.76025,S 2,T 35,E1 -4005.10214,E2 0,E3 0,E4 0,E5 0,E6 0}
; DECL LDAT LCPDATP123={VEL 1,ACC 100,APO_DIST 100,APO_FAC 50.0,ORI_TYP #VAR,CIRC_TYP #BASE,JERK_FAC 50.0}
DECL FDAT FP686={TOOL_NO 0,BASE_NO 0,IPO_FRAME #BASE,POINT2[] " ",TQ_STATE FALSE}
DECL E6POS XP686={X 12607.03936,Y -538.48386,Z 3940.5062,A -83.4604,B -12.81532,C -0.94267,S 2,T 35,E1 -10812.08896,E2 0,E3 0,E4 0,E5 0,E6 0}
; DECL LDAT LCPDATP124={VEL 1,ACC 100,APO_DIST 100,APO_FAC 50.0,ORI_TYP #VAR,CIRC_TYP #BASE,JERK_FAC 50.0}
DECL FDAT FP687={TOOL_NO 0,BASE_NO 0,IPO_FRAME #BASE,POINT2[] " ",TQ_STATE FALSE}
DECL E6POS XP687={X 12329.73693,Y -538.48386,Z 3940.5062,A -83.38777,B -15.32829,C -1.2413,S 2,T 35,E1 -10812.08896,E2 0,E3 0,E4 0,E5 0,E6 0}
; DECL LDAT LCPDATP130={VEL 1,ACC 100,APO_DIST 100,APO_FAC 50.0,ORI_TYP #VAR,CIRC_TYP #BASE,JERK_FAC 50.0}
DECL FDAT FP688={TOOL_NO 0,BASE_NO 0,IPO_FRAME #BASE,POINT2[] " ",TQ_STATE FALSE}
DECL E6POS XP688={X 6035.27715,Y -717.10158,Z 4003.70466,A -106.51042,B 6.34838,C 5.00917,S 2,T 35,E1 -4231.81368,E2 0,E3 0,E4 0,E5 0,E6 0}
; DECL LDAT LCPDATP131={VEL 1,ACC 100,APO_DIST 100,APO_FAC 50.0,ORI_TYP #VAR,CIRC_TYP #BASE,JERK_FAC 50.0}
DECL FDAT FP689={TOOL_NO 0,BASE_NO 0,IPO_FRAME #BASE,POINT2[] " ",TQ_STATE FALSE}
DECL E6POS XP689={X 6001.84737,Y -717.10113,Z 4003.70421,A -106.4599,B 4.5615,C 5.54032,S 2,T 35,E1 -4198.38336,E2 0,E3 0,E4 0,E5 0,E6 0}
; DECL LDAT LCPDATP125={VEL 1,ACC 100,APO_DIST 100,APO_FAC 50.0,ORI_TYP #VAR,CIRC_TYP #BASE,JERK_FAC 50.0}
DECL FDAT FP690={TOOL_NO 0,BASE_NO 0,IPO_FRAME #BASE,POINT2[] " ",TQ_STATE FALSE}
DECL E6POS XP690={X 12327.62864,Y -538.48366,Z 3940.50597,A -87.76623,B -17.49847,C -1.50503,S 2,T 35,E1 -10473.34117,E2 0,E3 0,E4 0,E5 0,E6 0}
; DECL LDAT LCPDATP126={VEL 1,ACC 100,APO_DIST 100,APO_FAC 50.0,ORI_TYP #VAR,CIRC_TYP #BASE,JERK_FAC 50.0}
DECL FDAT FP691={TOOL_NO 0,BASE_NO 0,IPO_FRAME #BASE,POINT2[] " ",TQ_STATE FALSE}
DECL E6POS XP691={X 12344.44126,Y -538.48354,Z 3940.50612,A -92.12133,B -19.55447,C -1.59012,S 2,T 35,E1 -10490.15446,E2 0,E3 0,E4 0,E5 0,E6 0}
; DECL LDAT LCPDATP132={VEL 1,ACC 100,APO_DIST 100,APO_FAC 50.0,ORI_TYP #VAR,CIRC_TYP #BASE,JERK_FAC 50.0}
DECL FDAT FP692={TOOL_NO 0,BASE_NO 0,IPO_FRAME #BASE,POINT2[] " ",TQ_STATE FALSE}
DECL E6POS XP692={X 5984.60315,Y -717.10142,Z 4003.7045,A -107.27293,B 2.66443,C 6.10126,S 2,T 35,E1 -4181.13976,E2 0,E3 0,E4 0,E5 0,E6 0}
; DECL LDAT LCPDATP133={VEL 1,ACC 100,APO_DIST 100,APO_FAC 50.0,ORI_TYP #VAR,CIRC_TYP #BASE,JERK_FAC 50.0}
DECL FDAT FP693={TOOL_NO 0,BASE_NO 0,IPO_FRAME #BASE,POINT2[] " ",TQ_STATE FALSE}
DECL E6POS XP693={X 5959.53065,Y -717.10165,Z 4003.70439,A -107.25516,B 0.74219,C 6.69889,S 2,T 35,E1 -4156.06702,E2 0,E3 0,E4 0,E5 0,E6 0}
; DECL LDAT LCPDATP127={VEL 1,ACC 100,APO_DIST 100,APO_FAC 50.0,ORI_TYP #VAR,CIRC_TYP #BASE,JERK_FAC 50.0}
DECL FDAT FP694={TOOL_NO 0,BASE_NO 0,IPO_FRAME #BASE,POINT2[] " ",TQ_STATE FALSE}
DECL E6POS XP694={X 12327.65948,Y -538.48376,Z 3940.50627,A -96.02004,B -21.56802,C -1.50992,S 2,T 35,E1 -10473.37259,E2 0,E3 0,E4 0,E5 0,E6 0}
; DECL LDAT LCPDATP128={VEL 1,ACC 100,APO_DIST 100,APO_FAC 50.0,ORI_TYP #VAR,CIRC_TYP #BASE,JERK_FAC 50.0}
DECL FDAT FP695={TOOL_NO 0,BASE_NO 0,IPO_FRAME #BASE,POINT2[] " ",TQ_STATE FALSE}
DECL E6POS XP695={X 12434.40962,Y -538.48361,Z 3791.38491,A -100.48203,B -23.59142,C -1.27711,S 2,T 35,E1 -10580.12251,E2 0,E3 0,E4 0,E5 0,E6 0}
; DECL LDAT LCPDATP134={VEL 1,ACC 100,APO_DIST 100,APO_FAC 50.0,ORI_TYP #VAR,CIRC_TYP #BASE,JERK_FAC 50.0}
DECL FDAT FP696={TOOL_NO 0,BASE_NO 0,IPO_FRAME #BASE,POINT2[] " ",TQ_STATE FALSE}
DECL E6POS XP696={X 6027.18413,Y -717.10157,Z 4003.70451,A -108.83879,B -1.2655,C 7.3225,S 2,T 35,E1 -4223.72032,E2 0,E3 0,E4 0,E5 0,E6 0}
; DECL LDAT LCPDATP135={VEL 1,ACC 100,APO_DIST 100,APO_FAC 50.0,ORI_TYP #VAR,CIRC_TYP #BASE,JERK_FAC 50.0}
DECL FDAT FP697={TOOL_NO 0,BASE_NO 0,IPO_FRAME #BASE,POINT2[] " ",TQ_STATE FALSE}
DECL E6POS XP697={X 5994.01853,Y -717.10159,Z 4003.70409,A -109.42003,B -3.44272,C 8.06654,S 2,T 35,E1 -4190.55423,E2 0,E3 0,E4 0,E5 0,E6 0}
; DECL LDAT LCPDATP129={VEL 1,ACC 100,APO_DIST 100,APO_FAC 50.0,ORI_TYP #VAR,CIRC_TYP #BASE,JERK_FAC 50.0}
DECL FDAT FP698={TOOL_NO 0,BASE_NO 0,IPO_FRAME #BASE,POINT2[] " ",TQ_STATE FALSE}
DECL E6POS XP698={X 12525.53957,Y -538.48385,Z 3733.39322,A -103.74147,B -24.12805,C -1.24549,S 2,T 35,E1 -10671.25219,E2 0,E3 0,E4 0,E5 0,E6 0}
; DECL LDAT LCPDATP138={VEL 1,ACC 100,APO_DIST 100,APO_FAC 50.0,ORI_TYP #VAR,CIRC_TYP #BASE,JERK_FAC 50.0}
DECL FDAT FP699={TOOL_NO 0,BASE_NO 0,IPO_FRAME #BASE,POINT2[] " ",TQ_STATE FALSE}
DECL E6POS XP699={X 12409.55634,Y -538.48385,Z 3733.39322,A -103.74147,B -24.12805,C -1.24549,S 2,T 35,E1 -10555.26896,E2 0,E3 0,E4 0,E5 0,E6 0}
; DECL LDAT LCPDATP136={VEL 1,ACC 100,APO_DIST 100,APO_FAC 50.0,ORI_TYP #VAR,CIRC_TYP #BASE,JERK_FAC 50.0}
DECL FDAT FP700={TOOL_NO 0,BASE_NO 0,IPO_FRAME #BASE,POINT2[] " ",TQ_STATE FALSE}
DECL E6POS XP700={X 5960.30101,Y -717.10136,Z 4003.70387,A -109.95564,B -5.51238,C 8.79955,S 2,T 35,E1 -4156.83652,E2 0,E3 0,E4 0,E5 0,E6 0}
; DECL LDAT LCPDATP137={VEL 1,ACC 100,APO_DIST 100,APO_FAC 50.0,ORI_TYP #VAR,CIRC_TYP #BASE,JERK_FAC 50.0}
DECL FDAT FP701={TOOL_NO 0,BASE_NO 0,IPO_FRAME #BASE,POINT2[] " ",TQ_STATE FALSE}
DECL E6POS XP701={X 5959.29294,Y -717.10098,Z 4003.70454,A -110.58224,B -7.77816,C 9.62993,S 2,T 35,E1 -4155.82897,E2 0,E3 0,E4 0,E5 0,E6 0}
; DECL LDAT LCPDATP139={VEL 1,ACC 100,APO_DIST 100,APO_FAC 50.0,ORI_TYP #VAR,CIRC_TYP #BASE,JERK_FAC 50.0}
DECL FDAT FP702={TOOL_NO 0,BASE_NO 0,IPO_FRAME #BASE,POINT2[] " ",TQ_STATE FALSE}
DECL E6POS XP702={X 12666.37592,Y -538.48386,Z 3733.39329,A -110.95703,B -23.34196,C -1.63568,S 2,T 35,E1 -10812.08896,E2 0,E3 0,E4 0,E5 0,E6 0}
; DECL LDAT LCPDATP140={VEL 1,ACC 100,APO_DIST 100,APO_FAC 50.0,ORI_TYP #VAR,CIRC_TYP #BASE,JERK_FAC 50.0}
DECL FDAT FP703={TOOL_NO 0,BASE_NO 0,IPO_FRAME #BASE,POINT2[] " ",TQ_STATE FALSE}
DECL E6POS XP703={X 12666.37592,Y -538.48386,Z 3700.25522,A -113.36831,B -23.34196,C -1.63568,S 2,T 35,E1 -10812.08896,E2 0,E3 0,E4 0,E5 0,E6 0}
; DECL LDAT LCPDATP149={VEL 1,ACC 100,APO_DIST 100,APO_FAC 50.0,ORI_TYP #VAR,CIRC_TYP #BASE,JERK_FAC 50.0}
DECL FDAT FP704={TOOL_NO 0,BASE_NO 0,IPO_FRAME #BASE,POINT2[] " ",TQ_STATE FALSE}
DECL E6POS XP704={X 5916.8006,Y -717.10155,Z 4003.70412,A -110.72224,B -10.13455,C 10.52896,S 2,T 35,E1 -4113.33656,E2 0,E3 0,E4 0,E5 0,E6 0}
; DECL LDAT LCPDATP150={VEL 1,ACC 100,APO_DIST 100,APO_FAC 50.0,ORI_TYP #VAR,CIRC_TYP #BASE,JERK_FAC 50.0}
DECL FDAT FP705={TOOL_NO 0,BASE_NO 0,IPO_FRAME #BASE,POINT2[] " ",TQ_STATE FALSE}
DECL E6POS XP705={X 5875.31565,Y -717.1012,Z 4003.70448,A -110.8879,B -12.32973,C 11.37928,S 2,T 35,E1 -4071.85169,E2 0,E3 0,E4 0,E5 0,E6 0}
; DECL LDAT LCPDATP141={VEL 1,ACC 100,APO_DIST 100,APO_FAC 50.0,ORI_TYP #VAR,CIRC_TYP #BASE,JERK_FAC 50.0}
DECL FDAT FP706={TOOL_NO 0,BASE_NO 0,IPO_FRAME #BASE,POINT2[] " ",TQ_STATE FALSE}
DECL E6POS XP706={X 12666.37592,Y -538.48386,Z 3675.40167,A -115.34787,B -23.34196,C -1.63568,S 2,T 35,E1 -10812.08896,E2 0,E3 0,E4 0,E5 0,E6 0}
; DECL LDAT LCPDATP142={VEL 1,ACC 100,APO_DIST 100,APO_FAC 50.0,ORI_TYP #VAR,CIRC_TYP #BASE,JERK_FAC 50.0}
DECL FDAT FP707={TOOL_NO 0,BASE_NO 0,IPO_FRAME #BASE,POINT2[] " ",TQ_STATE FALSE}
DECL E6POS XP707={X 12666.37592,Y -538.48386,Z 3725.10877,A -117.62399,B -22.31862,C -2.21953,S 2,T 35,E1 -10812.08896,E2 0,E3 0,E4 0,E5 0,E6 0}
; DECL LDAT LCPDATP151={VEL 1,ACC 100,APO_DIST 100,APO_FAC 50.0,ORI_TYP #VAR,CIRC_TYP #BASE,JERK_FAC 50.0}
DECL FDAT FP708={TOOL_NO 0,BASE_NO 0,IPO_FRAME #BASE,POINT2[] " ",TQ_STATE FALSE}
DECL E6POS XP708={X 5898.57722,Y -717.10122,Z 4003.70435,A -112.09203,B -14.38754,C 12.19033,S 2,T 35,E1 -4095.11298,E2 0,E3 0,E4 0,E5 0,E6 0}
; DECL LDAT LCPDATP152={VEL 1,ACC 100,APO_DIST 100,APO_FAC 50.0,ORI_TYP #VAR,CIRC_TYP #BASE,JERK_FAC 50.0}
DECL FDAT FP709={TOOL_NO 0,BASE_NO 0,IPO_FRAME #BASE,POINT2[] " ",TQ_STATE FALSE}
DECL E6POS XP709={X 5854.40488,Y -717.10171,Z 4003.70448,A -112.35649,B -16.71303,C 13.17652,S 2,T 35,E1 -4050.94133,E2 0,E3 0,E4 0,E5 0,E6 0}
; DECL LDAT LCPDATP143={VEL 1,ACC 100,APO_DIST 100,APO_FAC 50.0,ORI_TYP #VAR,CIRC_TYP #BASE,JERK_FAC 50.0}
DECL FDAT FP710={TOOL_NO 0,BASE_NO 0,IPO_FRAME #BASE,POINT2[] " ",TQ_STATE FALSE}
DECL E6POS XP710={X 12666.37592,Y -538.48386,Z 3708.53974,A -119.39266,B -22.0406,C -2.38888,S 2,T 35,E1 -10812.08896,E2 0,E3 0,E4 0,E5 0,E6 0}
; DECL LDAT LCPDATP144={VEL 1,ACC 100,APO_DIST 100,APO_FAC 50.0,ORI_TYP #VAR,CIRC_TYP #BASE,JERK_FAC 50.0}
DECL FDAT FP711={TOOL_NO 0,BASE_NO 0,IPO_FRAME #BASE,POINT2[] " ",TQ_STATE FALSE}
DECL E6POS XP711={X 12666.37592,Y -538.48386,Z 3716.82426,A -121.52366,B -21.70131,C -2.61349,S 2,T 35,E1 -10812.08896,E2 0,E3 0,E4 0,E5 0,E6 0}
; DECL LDAT LCPDATP153={VEL 1,ACC 100,APO_DIST 100,APO_FAC 50.0,ORI_TYP #VAR,CIRC_TYP #BASE,JERK_FAC 50.0}
DECL FDAT FP712={TOOL_NO 0,BASE_NO 0,IPO_FRAME #BASE,POINT2[] " ",TQ_STATE FALSE}
DECL E6POS XP712={X 5865.70091,Y -717.10124,Z 4003.70383,A -113.62634,B -18.80667,C 14.08679,S 2,T 35,E1 -4062.23613,E2 0,E3 0,E4 0,E5 0,E6 0}
; DECL LDAT LCPDATP154={VEL 1,ACC 100,APO_DIST 100,APO_FAC 50.0,ORI_TYP #VAR,CIRC_TYP #BASE,JERK_FAC 50.0}
DECL FDAT FP713={TOOL_NO 0,BASE_NO 0,IPO_FRAME #BASE,POINT2[] " ",TQ_STATE FALSE}
DECL E6POS XP713={X 5786.97193,Y -717.10138,Z 4003.70442,A -113.90846,B -20.59534,C 14.92344,S 2,T 35,E1 -3983.50839,E2 0,E3 0,E4 0,E5 0,E6 0}
; DECL LDAT LCPDATP145={VEL 1,ACC 100,APO_DIST 100,APO_FAC 50.0,ORI_TYP #VAR,CIRC_TYP #BASE,JERK_FAC 50.0}
DECL FDAT FP714={TOOL_NO 0,BASE_NO 0,IPO_FRAME #BASE,POINT2[] " ",TQ_STATE FALSE}
DECL E6POS XP714={X 12666.37592,Y -538.48386,Z 3691.97071,A -122.58569,B -21.70131,C -2.61349,S 2,T 35,E1 -10812.08896,E2 0,E3 0,E4 0,E5 0,E6 0}
; DECL LDAT LCPDATP146={VEL 1,ACC 100,APO_DIST 100,APO_FAC 50.0,ORI_TYP #VAR,CIRC_TYP #BASE,JERK_FAC 50.0}
DECL FDAT FP715={TOOL_NO 0,BASE_NO 0,IPO_FRAME #BASE,POINT2[] " ",TQ_STATE FALSE}
DECL E6POS XP715={X 12666.37592,Y -538.48386,Z 3741.67781,A -124.88801,B -20.60151,C -3.44033,S 2,T 35,E1 -10812.08896,E2 0,E3 0,E4 0,E5 0,E6 0}
; DECL LDAT LCPDATP155={VEL 1,ACC 100,APO_DIST 100,APO_FAC 50.0,ORI_TYP #VAR,CIRC_TYP #BASE,JERK_FAC 50.0}
DECL FDAT FP716={TOOL_NO 0,BASE_NO 0,IPO_FRAME #BASE,POINT2[] " ",TQ_STATE FALSE}
DECL E6POS XP716={X 5766.06143,Y -717.10078,Z 4003.7047,A -114.88478,B -21.82725,C 15.51221,S 2,T 35,E1 -3962.59803,E2 0,E3 0,E4 0,E5 0,E6 0}
; DECL LDAT LCPDATP156={VEL 1,ACC 100,APO_DIST 100,APO_FAC 50.0,ORI_TYP #VAR,CIRC_TYP #BASE,JERK_FAC 50.0}
DECL FDAT FP717={TOOL_NO 0,BASE_NO 0,IPO_FRAME #BASE,POINT2[] " ",TQ_STATE FALSE}
DECL E6POS XP717={X 5671.46198,Y -717.1018,Z 4003.704,A -116.65787,B -23.21109,C 16.21129,S 2,T 35,E1 -3867.99764,E2 0,E3 0,E4 0,E5 0,E6 0}
; DECL LDAT LCPDATP147={VEL 1,ACC 100,APO_DIST 100,APO_FAC 50.0,ORI_TYP #VAR,CIRC_TYP #BASE,JERK_FAC 50.0}
DECL FDAT FP718={TOOL_NO 0,BASE_NO 0,IPO_FRAME #BASE,POINT2[] " ",TQ_STATE FALSE}
DECL E6POS XP718={X 12666.37592,Y -538.48386,Z 3708.53974,A -127.07895,B -20.60151,C -3.44033,S 2,T 35,E1 -10812.08896,E2 0,E3 0,E4 0,E5 0,E6 0}
; DECL LDAT LCPDATP113={VEL 1,ACC 100,APO_DIST 100,APO_FAC 50.0,ORI_TYP #VAR,CIRC_TYP #BASE,JERK_FAC 50.0}
DECL FDAT FP719={TOOL_NO 0,BASE_NO 0,IPO_FRAME #BASE,POINT2[] " ",TQ_STATE FALSE}
DECL E6POS XP719={X 6379.94734,Y -681.40788,Z 3158.20554,A -102.40256,B 11.37187,C 4.81103,S 2,T 35,E1 -4209.91162,E2 0,E3 0,E4 0,E5 0,E6 0}
; DECL LDAT LCPDATP114={VEL 1,ACC 100,APO_DIST 100,APO_FAC 50.0,ORI_TYP #VAR,CIRC_TYP #BASE,JERK_FAC 50.0}
DECL FDAT FP720={TOOL_NO 0,BASE_NO 0,IPO_FRAME #BASE,POINT2[] " ",TQ_STATE FALSE}
DECL E6POS XP720={X 6328.481,Y -681.40737,Z 3158.20597,A -102.7078,B 7.77597,C 4.76025,S 2,T 35,E1 -4158.44503,E2 0,E3 0,E4 0,E5 0,E6 0}
; DECL LDAT LCPDATP115={VEL 1,ACC 100,APO_DIST 100,APO_FAC 50.0,ORI_TYP #VAR,CIRC_TYP #BASE,JERK_FAC 50.0}
DECL FDAT FP721={TOOL_NO 0,BASE_NO 0,IPO_FRAME #BASE,POINT2[] " ",TQ_STATE FALSE}
DECL E6POS XP721={X 12929.38089,Y -681.40737,Z 3158.20639,A -83.4604,B -12.81532,C -0.94267,S 2,T 35,E1 -10812.08896,E2 0,E3 0,E4 0,E5 0,E6 0}
; DECL LDAT LCPDATP116={VEL 1,ACC 100,APO_DIST 100,APO_FAC 50.0,ORI_TYP #VAR,CIRC_TYP #BASE,JERK_FAC 50.0}
DECL FDAT FP722={TOOL_NO 0,BASE_NO 0,IPO_FRAME #BASE,POINT2[] " ",TQ_STATE FALSE}
DECL E6POS XP722={X 12886.08572,Y -646.4113,Z 3336.02814,A -83.4604,B -12.81532,C -0.94267,S 2,T 35,E1 -10812.08896,E2 0,E3 0,E4 0,E5 0,E6 0}
; DECL LDAT LCPDATP117={VEL 1,ACC 100,APO_DIST 100,APO_FAC 50.0,ORI_TYP #VAR,CIRC_TYP #BASE,JERK_FAC 50.0}
DECL FDAT FP723={TOOL_NO 0,BASE_NO 0,IPO_FRAME #BASE,POINT2[] " ",TQ_STATE FALSE}
DECL E6POS XP723={X 6226.20694,Y -691.76303,Z 3410.82553,A -102.7078,B 7.77597,C 4.76022,S 2,T 35,E1 -4167.06683,E2 0,E3 0,E4 0,E5 0,E6 0}
; DECL LDAT LCPDATP118={VEL 1,ACC 100,APO_DIST 100,APO_FAC 50.0,ORI_TYP #VAR,CIRC_TYP #BASE,JERK_FAC 50.0}
DECL FDAT FP724={TOOL_NO 0,BASE_NO 0,IPO_FRAME #BASE,POINT2[] " ",TQ_STATE FALSE}
DECL E6POS XP724={X 6109.20944,Y -705.3695,Z 3654.40552,A -102.70779,B 7.77597,C 4.76025,S 2,T 35,E1 -4140.9372,E2 0,E3 0,E4 0,E5 0,E6 0}
; DECL LDAT LCPDATP121={VEL 1,ACC 100,APO_DIST 100,APO_FAC 50.0,ORI_TYP #VAR,CIRC_TYP #BASE,JERK_FAC 50.0}
DECL FDAT FP725={TOOL_NO 0,BASE_NO 0,IPO_FRAME #BASE,POINT2[] " ",TQ_STATE FALSE}
DECL E6POS XP725={X 12777.06723,Y -602.17839,Z 3573.69413,A -83.4604,B -12.81532,C -0.94267,S 2,T 35,E1 -10812.08896,E2 0,E3 0,E4 0,E5 0,E6 0}
; DECL LDAT LCPDATP122={VEL 1,ACC 100,APO_DIST 100,APO_FAC 50.0,ORI_TYP #VAR,CIRC_TYP #BASE,JERK_FAC 50.0}
DECL FDAT FP726={TOOL_NO 0,BASE_NO 0,IPO_FRAME #BASE,POINT2[] " ",TQ_STATE FALSE}
DECL E6POS XP726={X 12675.92788,Y -569.18264,Z 3775.2407,A -83.4604,B -12.81532,C -0.94267,S 2,T 35,E1 -10812.08896,E2 0,E3 0,E4 0,E5 0,E6 0}
; DECL LDAT LCPDATP119={VEL 1,ACC 100,APO_DIST 100,APO_FAC 50.0,ORI_TYP #VAR,CIRC_TYP #BASE,JERK_FAC 50.0}
DECL FDAT FP727={TOOL_NO 0,BASE_NO 0,IPO_FRAME #BASE,POINT2[] " ",TQ_STATE FALSE}
DECL E6POS XP727={X 6034.81499,Y -708.12179,Z 3847.76366,A -102.7078,B 7.77596,C 4.76026,S 2,T 35,E1 -4174.36752,E2 0,E3 0,E4 0,E5 0,E6 0}
; DECL LDAT LCPDATP120={VEL 1,ACC 100,APO_DIST 100,APO_FAC 50.0,ORI_TYP #VAR,CIRC_TYP #BASE,JERK_FAC 50.0}
DECL FDAT FP728={TOOL_NO 0,BASE_NO 0,IPO_FRAME #BASE,POINT2[] " ",TQ_STATE FALSE}
DECL E6POS XP728={X 5808.56571,Y -717.10091,Z 4003.7046,A -102.70779,B 7.77596,C 4.76025,S 2,T 35,E1 -4005.10214,E2 0,E3 0,E4 0,E5 0,E6 0}
; DECL LDAT LCPDATP123={VEL 1,ACC 100,APO_DIST 100,APO_FAC 50.0,ORI_TYP #VAR,CIRC_TYP #BASE,JERK_FAC 50.0}
DECL FDAT FP729={TOOL_NO 0,BASE_NO 0,IPO_FRAME #BASE,POINT2[] " ",TQ_STATE FALSE}
DECL E6POS XP729={X 12607.03936,Y -538.48386,Z 3940.5062,A -83.4604,B -12.81532,C -0.94267,S 2,T 35,E1 -10812.08896,E2 0,E3 0,E4 0,E5 0,E6 0}
; DECL LDAT LCPDATP124={VEL 1,ACC 100,APO_DIST 100,APO_FAC 50.0,ORI_TYP #VAR,CIRC_TYP #BASE,JERK_FAC 50.0}
DECL FDAT FP730={TOOL_NO 0,BASE_NO 0,IPO_FRAME #BASE,POINT2[] " ",TQ_STATE FALSE}
DECL E6POS XP730={X 12329.73693,Y -538.48386,Z 3940.5062,A -83.38777,B -15.32829,C -1.2413,S 2,T 35,E1 -10812.08896,E2 0,E3 0,E4 0,E5 0,E6 0}
; DECL LDAT LCPDATP130={VEL 1,ACC 100,APO_DIST 100,APO_FAC 50.0,ORI_TYP #VAR,CIRC_TYP #BASE,JERK_FAC 50.0}
DECL FDAT FP731={TOOL_NO 0,BASE_NO 0,IPO_FRAME #BASE,POINT2[] " ",TQ_STATE FALSE}
DECL E6POS XP731={X 6035.27715,Y -717.10158,Z 4003.70466,A -106.51042,B 6.34838,C 5.00917,S 2,T 35,E1 -4231.81368,E2 0,E3 0,E4 0,E5 0,E6 0}
; DECL LDAT LCPDATP131={VEL 1,ACC 100,APO_DIST 100,APO_FAC 50.0,ORI_TYP #VAR,CIRC_TYP #BASE,JERK_FAC 50.0}
DECL FDAT FP732={TOOL_NO 0,BASE_NO 0,IPO_FRAME #BASE,POINT2[] " ",TQ_STATE FALSE}
DECL E6POS XP732={X 6001.84737,Y -717.10113,Z 4003.70421,A -106.4599,B 4.5615,C 5.54032,S 2,T 35,E1 -4198.38336,E2 0,E3 0,E4 0,E5 0,E6 0}
; DECL LDAT LCPDATP125={VEL 1,ACC 100,APO_DIST 100,APO_FAC 50.0,ORI_TYP #VAR,CIRC_TYP #BASE,JERK_FAC 50.0}
DECL FDAT FP733={TOOL_NO 0,BASE_NO 0,IPO_FRAME #BASE,POINT2[] " ",TQ_STATE FALSE}
DECL E6POS XP733={X 12327.62864,Y -538.48366,Z 3940.50597,A -87.76623,B -17.49847,C -1.50503,S 2,T 35,E1 -10473.34117,E2 0,E3 0,E4 0,E5 0,E6 0}
; DECL LDAT LCPDATP126={VEL 1,ACC 100,APO_DIST 100,APO_FAC 50.0,ORI_TYP #VAR,CIRC_TYP #BASE,JERK_FAC 50.0}
DECL FDAT FP734={TOOL_NO 0,BASE_NO 0,IPO_FRAME #BASE,POINT2[] " ",TQ_STATE FALSE}
DECL E6POS XP734={X 12344.44126,Y -538.48354,Z 3940.50612,A -92.12133,B -19.55447,C -1.59012,S 2,T 35,E1 -10490.15446,E2 0,E3 0,E4 0,E5 0,E6 0}
; DECL LDAT LCPDATP132={VEL 1,ACC 100,APO_DIST 100,APO_FAC 50.0,ORI_TYP #VAR,CIRC_TYP #BASE,JERK_FAC 50.0}
DECL FDAT FP735={TOOL_NO 0,BASE_NO 0,IPO_FRAME #BASE,POINT2[] " ",TQ_STATE FALSE}
DECL E6POS XP735={X 5984.60315,Y -717.10142,Z 4003.7045,A -107.27293,B 2.66443,C 6.10126,S 2,T 35,E1 -4181.13976,E2 0,E3 0,E4 0,E5 0,E6 0}
; DECL LDAT LCPDATP133={VEL 1,ACC 100,APO_DIST 100,APO_FAC 50.0,ORI_TYP #VAR,CIRC_TYP #BASE,JERK_FAC 50.0}
DECL FDAT FP736={TOOL_NO 0,BASE_NO 0,IPO_FRAME #BASE,POINT2[] " ",TQ_STATE FALSE}
DECL E6POS XP736={X 5959.53065,Y -717.10165,Z 4003.70439,A -107.25516,B 0.74219,C 6.69889,S 2,T 35,E1 -4156.06702,E2 0,E3 0,E4 0,E5 0,E6 0}
; DECL LDAT LCPDATP127={VEL 1,ACC 100,APO_DIST 100,APO_FAC 50.0,ORI_TYP #VAR,CIRC_TYP #BASE,JERK_FAC 50.0}
DECL FDAT FP737={TOOL_NO 0,BASE_NO 0,IPO_FRAME #BASE,POINT2[] " ",TQ_STATE FALSE}
DECL E6POS XP737={X 12327.65948,Y -538.48376,Z 3940.50627,A -96.02004,B -21.56802,C -1.50992,S 2,T 35,E1 -10473.37259,E2 0,E3 0,E4 0,E5 0,E6 0}
; DECL LDAT LCPDATP128={VEL 1,ACC 100,APO_DIST 100,APO_FAC 50.0,ORI_TYP #VAR,CIRC_TYP #BASE,JERK_FAC 50.0}
DECL FDAT FP738={TOOL_NO 0,BASE_NO 0,IPO_FRAME #BASE,POINT2[] " ",TQ_STATE FALSE}
DECL E6POS XP738={X 12434.40962,Y -538.48361,Z 3791.38491,A -100.48203,B -23.59142,C -1.27711,S 2,T 35,E1 -10580.12251,E2 0,E3 0,E4 0,E5 0,E6 0}
; DECL LDAT LCPDATP134={VEL 1,ACC 100,APO_DIST 100,APO_FAC 50.0,ORI_TYP #VAR,CIRC_TYP #BASE,JERK_FAC 50.0}
DECL FDAT FP739={TOOL_NO 0,BASE_NO 0,IPO_FRAME #BASE,POINT2[] " ",TQ_STATE FALSE}
DECL E6POS XP739={X 6027.18413,Y -717.10157,Z 4003.70451,A -108.83879,B -1.2655,C 7.3225,S 2,T 35,E1 -4223.72032,E2 0,E3 0,E4 0,E5 0,E6 0}
; DECL LDAT LCPDATP135={VEL 1,ACC 100,APO_DIST 100,APO_FAC 50.0,ORI_TYP #VAR,CIRC_TYP #BASE,JERK_FAC 50.0}
DECL FDAT FP740={TOOL_NO 0,BASE_NO 0,IPO_FRAME #BASE,POINT2[] " ",TQ_STATE FALSE}
DECL E6POS XP740={X 5994.01853,Y -717.10159,Z 4003.70409,A -109.42003,B -3.44272,C 8.06654,S 2,T 35,E1 -4190.55423,E2 0,E3 0,E4 0,E5 0,E6 0}
; DECL LDAT LCPDATP129={VEL 1,ACC 100,APO_DIST 100,APO_FAC 50.0,ORI_TYP #VAR,CIRC_TYP #BASE,JERK_FAC 50.0}
DECL FDAT FP741={TOOL_NO 0,BASE_NO 0,IPO_FRAME #BASE,POINT2[] " ",TQ_STATE FALSE}
DECL E6POS XP741={X 12525.53957,Y -538.48385,Z 3733.39322,A -103.74147,B -24.12805,C -1.24549,S 2,T 35,E1 -10671.25219,E2 0,E3 0,E4 0,E5 0,E6 0}
; DECL LDAT LCPDATP138={VEL 1,ACC 100,APO_DIST 100,APO_FAC 50.0,ORI_TYP #VAR,CIRC_TYP #BASE,JERK_FAC 50.0}
DECL FDAT FP742={TOOL_NO 0,BASE_NO 0,IPO_FRAME #BASE,POINT2[] " ",TQ_STATE FALSE}
DECL E6POS XP742={X 12409.55634,Y -538.48385,Z 3733.39322,A -103.74147,B -24.12805,C -1.24549,S 2,T 35,E1 -10555.26896,E2 0,E3 0,E4 0,E5 0,E6 0}
; DECL LDAT LCPDATP136={VEL 1,ACC 100,APO_DIST 100,APO_FAC 50.0,ORI_TYP #VAR,CIRC_TYP #BASE,JERK_FAC 50.0}
DECL FDAT FP743={TOOL_NO 0,BASE_NO 0,IPO_FRAME #BASE,POINT2[] " ",TQ_STATE FALSE}
DECL E6POS XP743={X 5960.30101,Y -717.10136,Z 4003.70387,A -109.95564,B -5.51238,C 8.79955,S 2,T 35,E1 -4156.83652,E2 0,E3 0,E4 0,E5 0,E6 0}
; DECL LDAT LCPDATP137={VEL 1,ACC 100,APO_DIST 100,APO_FAC 50.0,ORI_TYP #VAR,CIRC_TYP #BASE,JERK_FAC 50.0}
DECL FDAT FP744={TOOL_NO 0,BASE_NO 0,IPO_FRAME #BASE,POINT2[] " ",TQ_STATE FALSE}
DECL E6POS XP744={X 5959.29294,Y -717.10098,Z 4003.70454,A -110.58224,B -7.77816,C 9.62993,S 2,T 35,E1 -4155.82897,E2 0,E3 0,E4 0,E5 0,E6 0}
; DECL LDAT LCPDATP139={VEL 1,ACC 100,APO_DIST 100,APO_FAC 50.0,ORI_TYP #VAR,CIRC_TYP #BASE,JERK_FAC 50.0}
DECL FDAT FP745={TOOL_NO 0,BASE_NO 0,IPO_FRAME #BASE,POINT2[] " ",TQ_STATE FALSE}
DECL E6POS XP745={X 12666.37592,Y -538.48386,Z 3733.39329,A -110.95703,B -23.34196,C -1.63568,S 2,T 35,E1 -10812.08896,E2 0,E3 0,E4 0,E5 0,E6 0}
; DECL LDAT LCPDATP140={VEL 1,ACC 100,APO_DIST 100,APO_FAC 50.0,ORI_TYP #VAR,CIRC_TYP #BASE,JERK_FAC 50.0}
DECL FDAT FP746={TOOL_NO 0,BASE_NO 0,IPO_FRAME #BASE,POINT2[] " ",TQ_STATE FALSE}
DECL E6POS XP746={X 12666.37592,Y -538.48386,Z 3700.25522,A -113.36831,B -23.34196,C -1.63568,S 2,T 35,E1 -10812.08896,E2 0,E3 0,E4 0,E5 0,E6 0}
; DECL LDAT LCPDATP149={VEL 1,ACC 100,APO_DIST 100,APO_FAC 50.0,ORI_TYP #VAR,CIRC_TYP #BASE,JERK_FAC 50.0}
DECL FDAT FP747={TOOL_NO 0,BASE_NO 0,IPO_FRAME #BASE,POINT2[] " ",TQ_STATE FALSE}
DECL E6POS XP747={X 5916.8006,Y -717.10155,Z 4003.70412,A -110.72224,B -10.13455,C 10.52896,S 2,T 35,E1 -4113.33656,E2 0,E3 0,E4 0,E5 0,E6 0}
; DECL LDAT LCPDATP150={VEL 1,ACC 100,APO_DIST 100,APO_FAC 50.0,ORI_TYP #VAR,CIRC_TYP #BASE,JERK_FAC 50.0}
DECL FDAT FP748={TOOL_NO 0,BASE_NO 0,IPO_FRAME #BASE,POINT2[] " ",TQ_STATE FALSE}
DECL E6POS XP748={X 5875.31565,Y -717.1012,Z 4003.70448,A -110.8879,B -12.32973,C 11.37928,S 2,T 35,E1 -4071.85169,E2 0,E3 0,E4 0,E5 0,E6 0}
; DECL LDAT LCPDATP141={VEL 1,ACC 100,APO_DIST 100,APO_FAC 50.0,ORI_TYP #VAR,CIRC_TYP #BASE,JERK_FAC 50.0}
DECL FDAT FP749={TOOL_NO 0,BASE_NO 0,IPO_FRAME #BASE,POINT2[] " ",TQ_STATE FALSE}
DECL E6POS XP749={X 12666.37592,Y -538.48386,Z 3675.40167,A -115.34787,B -23.34196,C -1.63568,S 2,T 35,E1 -10812.08896,E2 0,E3 0,E4 0,E5 0,E6 0}
; DECL LDAT LCPDATP142={VEL 1,ACC 100,APO_DIST 100,APO_FAC 50.0,ORI_TYP #VAR,CIRC_TYP #BASE,JERK_FAC 50.0}
DECL FDAT FP750={TOOL_NO 0,BASE_NO 0,IPO_FRAME #BASE,POINT2[] " ",TQ_STATE FALSE}
DECL E6POS XP750={X 12666.37592,Y -538.48386,Z 3725.10877,A -117.62399,B -22.31862,C -2.21953,S 2,T 35,E1 -10812.08896,E2 0,E3 0,E4 0,E5 0,E6 0}
; DECL LDAT LCPDATP151={VEL 1,ACC 100,APO_DIST 100,APO_FAC 50.0,ORI_TYP #VAR,CIRC_TYP #BASE,JERK_FAC 50.0}
DECL FDAT FP751={TOOL_NO 0,BASE_NO 0,IPO_FRAME #BASE,POINT2[] " ",TQ_STATE FALSE}
DECL E6POS XP751={X 5898.57722,Y -717.10122,Z 4003.70435,A -112.09203,B -14.38754,C 12.19033,S 2,T 35,E1 -4095.11298,E2 0,E3 0,E4 0,E5 0,E6 0}
; DECL LDAT LCPDATP152={VEL 1,ACC 100,APO_DIST 100,APO_FAC 50.0,ORI_TYP #VAR,CIRC_TYP #BASE,JERK_FAC 50.0}
DECL FDAT FP752={TOOL_NO 0,BASE_NO 0,IPO_FRAME #BASE,POINT2[] " ",TQ_STATE FALSE}
DECL E6POS XP752={X 5854.40488,Y -717.10171,Z 4003.70448,A -112.35649,B -16.71303,C 13.17652,S 2,T 35,E1 -4050.94133,E2 0,E3 0,E4 0,E5 0,E6 0}
; DECL LDAT LCPDATP143={VEL 1,ACC 100,APO_DIST 100,APO_FAC 50.0,ORI_TYP #VAR,CIRC_TYP #BASE,JERK_FAC 50.0}
DECL FDAT FP753={TOOL_NO 0,BASE_NO 0,IPO_FRAME #BASE,POINT2[] " ",TQ_STATE FALSE}
DECL E6POS XP753={X 12666.37592,Y -538.48386,Z 3708.53974,A -119.39266,B -22.0406,C -2.38888,S 2,T 35,E1 -10812.08896,E2 0,E3 0,E4 0,E5 0,E6 0}
; DECL LDAT LCPDATP144={VEL 1,ACC 100,APO_DIST 100,APO_FAC 50.0,ORI_TYP #VAR,CIRC_TYP #BASE,JERK_FAC 50.0}
DECL FDAT FP754={TOOL_NO 0,BASE_NO 0,IPO_FRAME #BASE,POINT2[] " ",TQ_STATE FALSE}
DECL E6POS XP754={X 12666.37592,Y -538.48386,Z 3716.82426,A -121.52366,B -21.70131,C -2.61349,S 2,T 35,E1 -10812.08896,E2 0,E3 0,E4 0,E5 0,E6 0}
; DECL LDAT LCPDATP153={VEL 1,ACC 100,APO_DIST 100,APO_FAC 50.0,ORI_TYP #VAR,CIRC_TYP #BASE,JERK_FAC 50.0}
DECL FDAT FP755={TOOL_NO 0,BASE_NO 0,IPO_FRAME #BASE,POINT2[] " ",TQ_STATE FALSE}
DECL E6POS XP755={X 5865.70091,Y -717.10124,Z 4003.70383,A -113.62634,B -18.80667,C 14.08679,S 2,T 35,E1 -4062.23613,E2 0,E3 0,E4 0,E5 0,E6 0}
; DECL LDAT LCPDATP154={VEL 1,ACC 100,APO_DIST 100,APO_FAC 50.0,ORI_TYP #VAR,CIRC_TYP #BASE,JERK_FAC 50.0}
DECL FDAT FP756={TOOL_NO 0,BASE_NO 0,IPO_FRAME #BASE,POINT2[] " ",TQ_STATE FALSE}
DECL E6POS XP756={X 5786.97193,Y -717.10138,Z 4003.70442,A -113.90846,B -20.59534,C 14.92344,S 2,T 35,E1 -3983.50839,E2 0,E3 0,E4 0,E5 0,E6 0}
; DECL LDAT LCPDATP145={VEL 1,ACC 100,APO_DIST 100,APO_FAC 50.0,ORI_TYP #VAR,CIRC_TYP #BASE,JERK_FAC 50.0}
DECL FDAT FP757={TOOL_NO 0,BASE_NO 0,IPO_FRAME #BASE,POINT2[] " ",TQ_STATE FALSE}
DECL E6POS XP757={X 12666.37592,Y -538.48386,Z 3691.97071,A -122.58569,B -21.70131,C -2.61349,S 2,T 35,E1 -10812.08896,E2 0,E3 0,E4 0,E5 0,E6 0}
; DECL LDAT LCPDATP146={VEL 1,ACC 100,APO_DIST 100,APO_FAC 50.0,ORI_TYP #VAR,CIRC_TYP #BASE,JERK_FAC 50.0}
DECL FDAT FP758={TOOL_NO 0,BASE_NO 0,IPO_FRAME #BASE,POINT2[] " ",TQ_STATE FALSE}
DECL E6POS XP758={X 12666.37592,Y -538.48386,Z 3741.67781,A -124.88801,B -20.60151,C -3.44033,S 2,T 35,E1 -10812.08896,E2 0,E3 0,E4 0,E5 0,E6 0}
; DECL LDAT LCPDATP155={VEL 1,ACC 100,APO_DIST 100,APO_FAC 50.0,ORI_TYP #VAR,CIRC_TYP #BASE,JERK_FAC 50.0}
DECL FDAT FP759={TOOL_NO 0,BASE_NO 0,IPO_FRAME #BASE,POINT2[] " ",TQ_STATE FALSE}
DECL E6POS XP759={X 5766.06143,Y -717.10078,Z 4003.7047,A -114.88478,B -21.82725,C 15.51221,S 2,T 35,E1 -3962.59803,E2 0,E3 0,E4 0,E5 0,E6 0}
; DECL LDAT LCPDATP156={VEL 1,ACC 100,APO_DIST 100,APO_FAC 50.0,ORI_TYP #VAR,CIRC_TYP #BASE,JERK_FAC 50.0}
DECL FDAT FP760={TOOL_NO 0,BASE_NO 0,IPO_FRAME #BASE,POINT2[] " ",TQ_STATE FALSE}
DECL E6POS XP760={X 5671.46198,Y -717.1018,Z 4003.704,A -116.65787,B -23.21109,C 16.21129,S 2,T 35,E1 -3867.99764,E2 0,E3 0,E4 0,E5 0,E6 0}
; DECL LDAT LCPDATP147={VEL 1,ACC 100,APO_DIST 100,APO_FAC 50.0,ORI_TYP #VAR,CIRC_TYP #BASE,JERK_FAC 50.0}
DECL FDAT FP761={TOOL_NO 0,BASE_NO 0,IPO_FRAME #BASE,POINT2[] " ",TQ_STATE FALSE}
DECL E6POS XP761={X 12666.37592,Y -538.48386,Z 3708.53974,A -127.07895,B -20.60151,C -3.44033,S 2,T 35,E1 -10812.08896,E2 0,E3 0,E4 0,E5 0,E6 0}
; DECL LDAT LCPDATP113={VEL 1,ACC 100,APO_DIST 100,APO_FAC 50.0,ORI_TYP #VAR,CIRC_TYP #BASE,JERK_FAC 50.0}
DECL FDAT FP762={TOOL_NO 0,BASE_NO 0,IPO_FRAME #BASE,POINT2[] " ",TQ_STATE FALSE}
DECL E6POS XP762={X 6379.94734,Y -681.40788,Z 3158.20554,A -102.40256,B 11.37187,C 4.81103,S 2,T 35,E1 -4209.91162,E2 0,E3 0,E4 0,E5 0,E6 0}
; DECL LDAT LCPDATP114={VEL 1,ACC 100,APO_DIST 100,APO_FAC 50.0,ORI_TYP #VAR,CIRC_TYP #BASE,JERK_FAC 50.0}
DECL FDAT FP763={TOOL_NO 0,BASE_NO 0,IPO_FRAME #BASE,POINT2[] " ",TQ_STATE FALSE}
DECL E6POS XP763={X 6328.481,Y -681.40737,Z 3158.20597,A -102.7078,B 7.77597,C 4.76025,S 2,T 35,E1 -4158.44503,E2 0,E3 0,E4 0,E5 0,E6 0}
; DECL LDAT LCPDATP115={VEL 1,ACC 100,APO_DIST 100,APO_FAC 50.0,ORI_TYP #VAR,CIRC_TYP #BASE,JERK_FAC 50.0}
DECL FDAT FP764={TOOL_NO 0,BASE_NO 0,IPO_FRAME #BASE,POINT2[] " ",TQ_STATE FALSE}
DECL E6POS XP764={X 12929.38089,Y -681.40737,Z 3158.20639,A -83.4604,B -12.81532,C -0.94267,S 2,T 35,E1 -10812.08896,E2 0,E3 0,E4 0,E5 0,E6 0}
; DECL LDAT LCPDATP116={VEL 1,ACC 100,APO_DIST 100,APO_FAC 50.0,ORI_TYP #VAR,CIRC_TYP #BASE,JERK_FAC 50.0}
DECL FDAT FP765={TOOL_NO 0,BASE_NO 0,IPO_FRAME #BASE,POINT2[] " ",TQ_STATE FALSE}
DECL E6POS XP765={X 12886.08572,Y -646.4113,Z 3336.02814,A -83.4604,B -12.81532,C -0.94267,S 2,T 35,E1 -10812.08896,E2 0,E3 0,E4 0,E5 0,E6 0}
; DECL LDAT LCPDATP117={VEL 1,ACC 100,APO_DIST 100,APO_FAC 50.0,ORI_TYP #VAR,CIRC_TYP #BASE,JERK_FAC 50.0}
DECL FDAT FP766={TOOL_NO 0,BASE_NO 0,IPO_FRAME #BASE,POINT2[] " ",TQ_STATE FALSE}
DECL E6POS XP766={X 6226.20694,Y -691.76303,Z 3410.82553,A -102.7078,B 7.77597,C 4.76022,S 2,T 35,E1 -4167.06683,E2 0,E3 0,E4 0,E5 0,E6 0}
; DECL LDAT LCPDATP118={VEL 1,ACC 100,APO_DIST 100,APO_FAC 50.0,ORI_TYP #VAR,CIRC_TYP #BASE,JERK_FAC 50.0}
DECL FDAT FP767={TOOL_NO 0,BASE_NO 0,IPO_FRAME #BASE,POINT2[] " ",TQ_STATE FALSE}
DECL E6POS XP767={X 6109.20944,Y -705.3695,Z 3654.40552,A -102.70779,B 7.77597,C 4.76025,S 2,T 35,E1 -4140.9372,E2 0,E3 0,E4 0,E5 0,E6 0}
; DECL LDAT LCPDATP121={VEL 1,ACC 100,APO_DIST 100,APO_FAC 50.0,ORI_TYP #VAR,CIRC_TYP #BASE,JERK_FAC 50.0}
DECL FDAT FP768={TOOL_NO 0,BASE_NO 0,IPO_FRAME #BASE,POINT2[] " ",TQ_STATE FALSE}
DECL E6POS XP768={X 12777.06723,Y -602.17839,Z 3573.69413,A -83.4604,B -12.81532,C -0.94267,S 2,T 35,E1 -10812.08896,E2 0,E3 0,E4 0,E5 0,E6 0}
; DECL LDAT LCPDATP122={VEL 1,ACC 100,APO_DIST 100,APO_FAC 50.0,ORI_TYP #VAR,CIRC_TYP #BASE,JERK_FAC 50.0}
DECL FDAT FP769={TOOL_NO 0,BASE_NO 0,IPO_FRAME #BASE,POINT2[] " ",TQ_STATE FALSE}
DECL E6POS XP769={X 12675.92788,Y -569.18264,Z 3775.2407,A -83.4604,B -12.81532,C -0.94267,S 2,T 35,E1 -10812.08896,E2 0,E3 0,E4 0,E5 0,E6 0}
; DECL LDAT LCPDATP119={VEL 1,ACC 100,APO_DIST 100,APO_FAC 50.0,ORI_TYP #VAR,CIRC_TYP #BASE,JERK_FAC 50.0}
DECL FDAT FP770={TOOL_NO 0,BASE_NO 0,IPO_FRAME #BASE,POINT2[] " ",TQ_STATE FALSE}
DECL E6POS XP770={X 6034.81499,Y -708.12179,Z 3847.76366,A -102.7078,B 7.77596,C 4.76026,S 2,T 35,E1 -4174.36752,E2 0,E3 0,E4 0,E5 0,E6 0}
; DECL LDAT LCPDATP120={VEL 1,ACC 100,APO_DIST 100,APO_FAC 50.0,ORI_TYP #VAR,CIRC_TYP #BASE,JERK_FAC 50.0}
DECL FDAT FP771={TOOL_NO 0,BASE_NO 0,IPO_FRAME #BASE,POINT2[] " ",TQ_STATE FALSE}
DECL E6POS XP771={X 5808.56571,Y -717.10091,Z 4003.7046,A -102.70779,B 7.77596,C 4.76025,S 2,T 35,E1 -4005.10214,E2 0,E3 0,E4 0,E5 0,E6 0}
; DECL LDAT LCPDATP123={VEL 1,ACC 100,APO_DIST 100,APO_FAC 50.0,ORI_TYP #VAR,CIRC_TYP #BASE,JERK_FAC 50.0}
DECL FDAT FP772={TOOL_NO 0,BASE_NO 0,IPO_FRAME #BASE,POINT2[] " ",TQ_STATE FALSE}
DECL E6POS XP772={X 12607.03936,Y -538.48386,Z 3940.5062,A -83.4604,B -12.81532,C -0.94267,S 2,T 35,E1 -10812.08896,E2 0,E3 0,E4 0,E5 0,E6 0}
; DECL LDAT LCPDATP124={VEL 1,ACC 100,APO_DIST 100,APO_FAC 50.0,ORI_TYP #VAR,CIRC_TYP #BASE,JERK_FAC 50.0}
DECL FDAT FP773={TOOL_NO 0,BASE_NO 0,IPO_FRAME #BASE,POINT2[] " ",TQ_STATE FALSE}
DECL E6POS XP773={X 12329.73693,Y -538.48386,Z 3940.5062,A -83.38777,B -15.32829,C -1.2413,S 2,T 35,E1 -10812.08896,E2 0,E3 0,E4 0,E5 0,E6 0}
; DECL LDAT LCPDATP130={VEL 1,ACC 100,APO_DIST 100,APO_FAC 50.0,ORI_TYP #VAR,CIRC_TYP #BASE,JERK_FAC 50.0}
DECL FDAT FP774={TOOL_NO 0,BASE_NO 0,IPO_FRAME #BASE,POINT2[] " ",TQ_STATE FALSE}
DECL E6POS XP774={X 6035.27715,Y -717.10158,Z 4003.70466,A -106.51042,B 6.34838,C 5.00917,S 2,T 35,E1 -4231.81368,E2 0,E3 0,E4 0,E5 0,E6 0}
; DECL LDAT LCPDATP131={VEL 1,ACC 100,APO_DIST 100,APO_FAC 50.0,ORI_TYP #VAR,CIRC_TYP #BASE,JERK_FAC 50.0}
DECL FDAT FP775={TOOL_NO 0,BASE_NO 0,IPO_FRAME #BASE,POINT2[] " ",TQ_STATE FALSE}
DECL E6POS XP775={X 6001.84737,Y -717.10113,Z 4003.70421,A -106.4599,B 4.5615,C 5.54032,S 2,T 35,E1 -4198.38336,E2 0,E3 0,E4 0,E5 0,E6 0}
; DECL LDAT LCPDATP125={VEL 1,ACC 100,APO_DIST 100,APO_FAC 50.0,ORI_TYP #VAR,CIRC_TYP #BASE,JERK_FAC 50.0}
DECL FDAT FP776={TOOL_NO 0,BASE_NO 0,IPO_FRAME #BASE,POINT2[] " ",TQ_STATE FALSE}
DECL E6POS XP776={X 12327.62864,Y -538.48366,Z 3940.50597,A -87.76623,B -17.49847,C -1.50503,S 2,T 35,E1 -10473.34117,E2 0,E3 0,E4 0,E5 0,E6 0}
; DECL LDAT LCPDATP126={VEL 1,ACC 100,APO_DIST 100,APO_FAC 50.0,ORI_TYP #VAR,CIRC_TYP #BASE,JERK_FAC 50.0}
DECL FDAT FP777={TOOL_NO 0,BASE_NO 0,IPO_FRAME #BASE,POINT2[] " ",TQ_STATE FALSE}
DECL E6POS XP777={X 12344.44126,Y -538.48354,Z 3940.50612,A -92.12133,B -19.55447,C -1.59012,S 2,T 35,E1 -10490.15446,E2 0,E3 0,E4 0,E5 0,E6 0}
; DECL LDAT LCPDATP132={VEL 1,ACC 100,APO_DIST 100,APO_FAC 50.0,ORI_TYP #VAR,CIRC_TYP #BASE,JERK_FAC 50.0}
DECL FDAT FP778={TOOL_NO 0,BASE_NO 0,IPO_FRAME #BASE,POINT2[] " ",TQ_STATE FALSE}
DECL E6POS XP778={X 5984.60315,Y -717.10142,Z 4003.7045,A -107.27293,B 2.66443,C 6.10126,S 2,T 35,E1 -4181.13976,E2 0,E3 0,E4 0,E5 0,E6 0}
; DECL LDAT LCPDATP133={VEL 1,ACC 100,APO_DIST 100,APO_FAC 50.0,ORI_TYP #VAR,CIRC_TYP #BASE,JERK_FAC 50.0}
DECL FDAT FP779={TOOL_NO 0,BASE_NO 0,IPO_FRAME #BASE,POINT2[] " ",TQ_STATE FALSE}
DECL E6POS XP779={X 5959.53065,Y -717.10165,Z 4003.70439,A -107.25516,B 0.74219,C 6.69889,S 2,T 35,E1 -4156.06702,E2 0,E3 0,E4 0,E5 0,E6 0}
; DECL LDAT LCPDATP127={VEL 1,ACC 100,APO_DIST 100,APO_FAC 50.0,ORI_TYP #VAR,CIRC_TYP #BASE,JERK_FAC 50.0}
DECL FDAT FP780={TOOL_NO 0,BASE_NO 0,IPO_FRAME #BASE,POINT2[] " ",TQ_STATE FALSE}
DECL E6POS XP780={X 12327.65948,Y -538.48376,Z 3940.50627,A -96.02004,B -21.56802,C -1.50992,S 2,T 35,E1 -10473.37259,E2 0,E3 0,E4 0,E5 0,E6 0}
; DECL LDAT LCPDATP128={VEL 1,ACC 100,APO_DIST 100,APO_FAC 50.0,ORI_TYP #VAR,CIRC_TYP #BASE,JERK_FAC 50.0}
DECL FDAT FP781={TOOL_NO 0,BASE_NO 0,IPO_FRAME #BASE,POINT2[] " ",TQ_STATE FALSE}
DECL E6POS XP781={X 12434.40962,Y -538.48361,Z 3791.38491,A -100.48203,B -23.59142,C -1.27711,S 2,T 35,E1 -10580.12251,E2 0,E3 0,E4 0,E5 0,E6 0}
; DECL LDAT LCPDATP134={VEL 1,ACC 100,APO_DIST 100,APO_FAC 50.0,ORI_TYP #VAR,CIRC_TYP #BASE,JERK_FAC 50.0}
DECL FDAT FP782={TOOL_NO 0,BASE_NO 0,IPO_FRAME #BASE,POINT2[] " ",TQ_STATE FALSE}
DECL E6POS XP782={X 6027.18413,Y -717.10157,Z 4003.70451,A -108.83879,B -1.2655,C 7.3225,S 2,T 35,E1 -4223.72032,E2 0,E3 0,E4 0,E5 0,E6 0}
; DECL LDAT LCPDATP135={VEL 1,ACC 100,APO_DIST 100,APO_FAC 50.0,ORI_TYP #VAR,CIRC_TYP #BASE,JERK_FAC 50.0}
DECL FDAT FP783={TOOL_NO 0,BASE_NO 0,IPO_FRAME #BASE,POINT2[] " ",TQ_STATE FALSE}
DECL E6POS XP783={X 5994.01853,Y -717.10159,Z 4003.70409,A -109.42003,B -3.44272,C 8.06654,S 2,T 35,E1 -4190.55423,E2 0,E3 0,E4 0,E5 0,E6 0}
; DECL LDAT LCPDATP129={VEL 1,ACC 100,APO_DIST 100,APO_FAC 50.0,ORI_TYP #VAR,CIRC_TYP #BASE,JERK_FAC 50.0}
DECL FDAT FP784={TOOL_NO 0,BASE_NO 0,IPO_FRAME #BASE,POINT2[] " ",TQ_STATE FALSE}
DECL E6POS XP784={X 12525.53957,Y -538.48385,Z 3733.39322,A -103.74147,B -24.12805,C -1.24549,S 2,T 35,E1 -10671.25219,E2 0,E3 0,E4 0,E5 0,E6 0}
; DECL LDAT LCPDATP138={VEL 1,ACC 100,APO_DIST 100,APO_FAC 50.0,ORI_TYP #VAR,CIRC_TYP #BASE,JERK_FAC 50.0}
DECL FDAT FP785={TOOL_NO 0,BASE_NO 0,IPO_FRAME #BASE,POINT2[] " ",TQ_STATE FALSE}
DECL E6POS XP785={X 12409.55634,Y -538.48385,Z 3733.39322,A -103.74147,B -24.12805,C -1.24549,S 2,T 35,E1 -10555.26896,E2 0,E3 0,E4 0,E5 0,E6 0}
; DECL LDAT LCPDATP136={VEL 1,ACC 100,APO_DIST 100,APO_FAC 50.0,ORI_TYP #VAR,CIRC_TYP #BASE,JERK_FAC 50.0}
DECL FDAT FP786={TOOL_NO 0,BASE_NO 0,IPO_FRAME #BASE,POINT2[] " ",TQ_STATE FALSE}
DECL E6POS XP786={X 5960.30101,Y -717.10136,Z 4003.70387,A -109.95564,B -5.51238,C 8.79955,S 2,T 35,E1 -4156.83652,E2 0,E3 0,E4 0,E5 0,E6 0}
; DECL LDAT LCPDATP137={VEL 1,ACC 100,APO_DIST 100,APO_FAC 50.0,ORI_TYP #VAR,CIRC_TYP #BASE,JERK_FAC 50.0}
DECL FDAT FP787={TOOL_NO 0,BASE_NO 0,IPO_FRAME #BASE,POINT2[] " ",TQ_STATE FALSE}
DECL E6POS XP787={X 5959.29294,Y -717.10098,Z 4003.70454,A -110.58224,B -7.77816,C 9.62993,S 2,T 35,E1 -4155.82897,E2 0,E3 0,E4 0,E5 0,E6 0}
; DECL LDAT LCPDATP139={VEL 1,ACC 100,APO_DIST 100,APO_FAC 50.0,ORI_TYP #VAR,CIRC_TYP #BASE,JERK_FAC 50.0}
DECL FDAT FP788={TOOL_NO 0,BASE_NO 0,IPO_FRAME #BASE,POINT2[] " ",TQ_STATE FALSE}
DECL E6POS XP788={X 12666.37592,Y -538.48386,Z 3733.39329,A -110.95703,B -23.34196,C -1.63568,S 2,T 35,E1 -10812.08896,E2 0,E3 0,E4 0,E5 0,E6 0}
; DECL LDAT LCPDATP140={VEL 1,ACC 100,APO_DIST 100,APO_FAC 50.0,ORI_TYP #VAR,CIRC_TYP #BASE,JERK_FAC 50.0}
DECL FDAT FP789={TOOL_NO 0,BASE_NO 0,IPO_FRAME #BASE,POINT2[] " ",TQ_STATE FALSE}
DECL E6POS XP789={X 12666.37592,Y -538.48386,Z 3700.25522,A -113.36831,B -23.34196,C -1.63568,S 2,T 35,E1 -10812.08896,E2 0,E3 0,E4 0,E5 0,E6 0}
; DECL LDAT LCPDATP149={VEL 1,ACC 100,APO_DIST 100,APO_FAC 50.0,ORI_TYP #VAR,CIRC_TYP #BASE,JERK_FAC 50.0}
DECL FDAT FP790={TOOL_NO 0,BASE_NO 0,IPO_FRAME #BASE,POINT2[] " ",TQ_STATE FALSE}
DECL E6POS XP790={X 5916.8006,Y -717.10155,Z 4003.70412,A -110.72224,B -10.13455,C 10.52896,S 2,T 35,E1 -4113.33656,E2 0,E3 0,E4 0,E5 0,E6 0}
; DECL LDAT LCPDATP150={VEL 1,ACC 100,APO_DIST 100,APO_FAC 50.0,ORI_TYP #VAR,CIRC_TYP #BASE,JERK_FAC 50.0}
DECL FDAT FP791={TOOL_NO 0,BASE_NO 0,IPO_FRAME #BASE,POINT2[] " ",TQ_STATE FALSE}
DECL E6POS XP791={X 5875.31565,Y -717.1012,Z 4003.70448,A -110.8879,B -12.32973,C 11.37928,S 2,T 35,E1 -4071.85169,E2 0,E3 0,E4 0,E5 0,E6 0}
; DECL LDAT LCPDATP141={VEL 1,ACC 100,APO_DIST 100,APO_FAC 50.0,ORI_TYP #VAR,CIRC_TYP #BASE,JERK_FAC 50.0}
DECL FDAT FP792={TOOL_NO 0,BASE_NO 0,IPO_FRAME #BASE,POINT2[] " ",TQ_STATE FALSE}
DECL E6POS XP792={X 12666.37592,Y -538.48386,Z 3675.40167,A -115.34787,B -23.34196,C -1.63568,S 2,T 35,E1 -10812.08896,E2 0,E3 0,E4 0,E5 0,E6 0}
; DECL LDAT LCPDATP142={VEL 1,ACC 100,APO_DIST 100,APO_FAC 50.0,ORI_TYP #VAR,CIRC_TYP #BASE,JERK_FAC 50.0}
DECL FDAT FP793={TOOL_NO 0,BASE_NO 0,IPO_FRAME #BASE,POINT2[] " ",TQ_STATE FALSE}
DECL E6POS XP793={X 12666.37592,Y -538.48386,Z 3725.10877,A -117.62399,B -22.31862,C -2.21953,S 2,T 35,E1 -10812.08896,E2 0,E3 0,E4 0,E5 0,E6 0}
; DECL LDAT LCPDATP151={VEL 1,ACC 100,APO_DIST 100,APO_FAC 50.0,ORI_TYP #VAR,CIRC_TYP #BASE,JERK_FAC 50.0}
DECL FDAT FP794={TOOL_NO 0,BASE_NO 0,IPO_FRAME #BASE,POINT2[] " ",TQ_STATE FALSE}
DECL E6POS XP794={X 5898.57722,Y -717.10122,Z 4003.70435,A -112.09203,B -14.38754,C 12.19033,S 2,T 35,E1 -4095.11298,E2 0,E3 0,E4 0,E5 0,E6 0}
; DECL LDAT LCPDATP152={VEL 1,ACC 100,APO_DIST 100,APO_FAC 50.0,ORI_TYP #VAR,CIRC_TYP #BASE,JERK_FAC 50.0}
DECL FDAT FP795={TOOL_NO 0,BASE_NO 0,IPO_FRAME #BASE,POINT2[] " ",TQ_STATE FALSE}
DECL E6POS XP795={X 5854.40488,Y -717.10171,Z 4003.70448,A -112.35649,B -16.71303,C 13.17652,S 2,T 35,E1 -4050.94133,E2 0,E3 0,E4 0,E5 0,E6 0}
; DECL LDAT LCPDATP143={VEL 1,ACC 100,APO_DIST 100,APO_FAC 50.0,ORI_TYP #VAR,CIRC_TYP #BASE,JERK_FAC 50.0}
DECL FDAT FP796={TOOL_NO 0,BASE_NO 0,IPO_FRAME #BASE,POINT2[] " ",TQ_STATE FALSE}
DECL E6POS XP796={X 12666.37592,Y -538.48386,Z 3708.53974,A -119.39266,B -22.0406,C -2.38888,S 2,T 35,E1 -10812.08896,E2 0,E3 0,E4 0,E5 0,E6 0}
; DECL LDAT LCPDATP144={VEL 1,ACC 100,APO_DIST 100,APO_FAC 50.0,ORI_TYP #VAR,CIRC_TYP #BASE,JERK_FAC 50.0}
DECL FDAT FP797={TOOL_NO 0,BASE_NO 0,IPO_FRAME #BASE,POINT2[] " ",TQ_STATE FALSE}
DECL E6POS XP797={X 12666.37592,Y -538.48386,Z 3716.82426,A -121.52366,B -21.70131,C -2.61349,S 2,T 35,E1 -10812.08896,E2 0,E3 0,E4 0,E5 0,E6 0}
; DECL LDAT LCPDATP153={VEL 1,ACC 100,APO_DIST 100,APO_FAC 50.0,ORI_TYP #VAR,CIRC_TYP #BASE,JERK_FAC 50.0}
DECL FDAT FP798={TOOL_NO 0,BASE_NO 0,IPO_FRAME #BASE,POINT2[] " ",TQ_STATE FALSE}
DECL E6POS XP798={X 5865.70091,Y -717.10124,Z 4003.70383,A -113.62634,B -18.80667,C 14.08679,S 2,T 35,E1 -4062.23613,E2 0,E3 0,E4 0,E5 0,E6 0}
; DECL LDAT LCPDATP154={VEL 1,ACC 100,APO_DIST 100,APO_FAC 50.0,ORI_TYP #VAR,CIRC_TYP #BASE,JERK_FAC 50.0}
DECL FDAT FP799={TOOL_NO 0,BASE_NO 0,IPO_FRAME #BASE,POINT2[] " ",TQ_STATE FALSE}
DECL E6POS XP799={X 5786.97193,Y -717.10138,Z 4003.70442,A -113.90846,B -20.59534,C 14.92344,S 2,T 35,E1 -3983.50839,E2 0,E3 0,E4 0,E5 0,E6 0}
; DECL LDAT LCPDATP145={VEL 1,ACC 100,APO_DIST 100,APO_FAC 50.0,ORI_TYP #VAR,CIRC_TYP #BASE,JERK_FAC 50.0}
DECL FDAT FP800={TOOL_NO 0,BASE_NO 0,IPO_FRAME #BASE,POINT2[] " ",TQ_STATE FALSE}
DECL E6POS XP800={X 12666.37592,Y -538.48386,Z 3691.97071,A -122.58569,B -21.70131,C -2.61349,S 2,T 35,E1 -10812.08896,E2 0,E3 0,E4 0,E5 0,E6 0}
; DECL LDAT LCPDATP146={VEL 1,ACC 100,APO_DIST 100,APO_FAC 50.0,ORI_TYP #VAR,CIRC_TYP #BASE,JERK_FAC 50.0}
DECL FDAT FP801={TOOL_NO 0,BASE_NO 0,IPO_FRAME #BASE,POINT2[] " ",TQ_STATE FALSE}
DECL E6POS XP801={X 12666.37592,Y -538.48386,Z 3741.67781,A -124.88801,B -20.60151,C -3.44033,S 2,T 35,E1 -10812.08896,E2 0,E3 0,E4 0,E5 0,E6 0}
; DECL LDAT LCPDATP155={VEL 1,ACC 100,APO_DIST 100,APO_FAC 50.0,ORI_TYP #VAR,CIRC_TYP #BASE,JERK_FAC 50.0}
DECL FDAT FP802={TOOL_NO 0,BASE_NO 0,IPO_FRAME #BASE,POINT2[] " ",TQ_STATE FALSE}
DECL E6POS XP802={X 5766.06143,Y -717.10078,Z 4003.7047,A -114.88478,B -21.82725,C 15.51221,S 2,T 35,E1 -3962.59803,E2 0,E3 0,E4 0,E5 0,E6 0}
; DECL LDAT LCPDATP156={VEL 1,ACC 100,APO_DIST 100,APO_FAC 50.0,ORI_TYP #VAR,CIRC_TYP #BASE,JERK_FAC 50.0}
DECL FDAT FP803={TOOL_NO 0,BASE_NO 0,IPO_FRAME #BASE,POINT2[] " ",TQ_STATE FALSE}
DECL E6POS XP803={X 5671.46198,Y -717.1018,Z 4003.704,A -116.65787,B -23.21109,C 16.21129,S 2,T 35,E1 -3867.99764,E2 0,E3 0,E4 0,E5 0,E6 0}
; DECL LDAT LCPDATP147={VEL 1,ACC 100,APO_DIST 100,APO_FAC 50.0,ORI_TYP #VAR,CIRC_TYP #BASE,JERK_FAC 50.0}
DECL FDAT FP804={TOOL_NO 0,BASE_NO 0,IPO_FRAME #BASE,POINT2[] " ",TQ_STATE FALSE}
DECL E6POS XP804={X 12666.37592,Y -538.48386,Z 3708.53974,A -127.07895,B -20.60151,C -3.44033,S 2,T 35,E1 -10812.08896,E2 0,E3 0,E4 0,E5 0,E6 0}
; DECL LDAT LCPDATP113={VEL 1,ACC 100,APO_DIST 100,APO_FAC 50.0,ORI_TYP #VAR,CIRC_TYP #BASE,JERK_FAC 50.0}
DECL FDAT FP805={TOOL_NO 0,BASE_NO 0,IPO_FRAME #BASE,POINT2[] " ",TQ_STATE FALSE}
DECL E6POS XP805={X 6379.94734,Y -681.40788,Z 3158.20554,A -102.40256,B 11.37187,C 4.81103,S 2,T 35,E1 -4209.91162,E2 0,E3 0,E4 0,E5 0,E6 0}
; DECL LDAT LCPDATP114={VEL 1,ACC 100,APO_DIST 100,APO_FAC 50.0,ORI_TYP #VAR,CIRC_TYP #BASE,JERK_FAC 50.0}
DECL FDAT FP806={TOOL_NO 0,BASE_NO 0,IPO_FRAME #BASE,POINT2[] " ",TQ_STATE FALSE}
DECL E6POS XP806={X 6328.481,Y -681.40737,Z 3158.20597,A -102.7078,B 7.77597,C 4.76025,S 2,T 35,E1 -4158.44503,E2 0,E3 0,E4 0,E5 0,E6 0}
; DECL LDAT LCPDATP115={VEL 1,ACC 100,APO_DIST 100,APO_FAC 50.0,ORI_TYP #VAR,CIRC_TYP #BASE,JERK_FAC 50.0}
DECL FDAT FP807={TOOL_NO 0,BASE_NO 0,IPO_FRAME #BASE,POINT2[] " ",TQ_STATE FALSE}
DECL E6POS XP807={X 12929.38089,Y -681.40737,Z 3158.20639,A -83.4604,B -12.81532,C -0.94267,S 2,T 35,E1 -10812.08896,E2 0,E3 0,E4 0,E5 0,E6 0}
; DECL LDAT LCPDATP116={VEL 1,ACC 100,APO_DIST 100,APO_FAC 50.0,ORI_TYP #VAR,CIRC_TYP #BASE,JERK_FAC 50.0}
DECL FDAT FP808={TOOL_NO 0,BASE_NO 0,IPO_FRAME #BASE,POINT2[] " ",TQ_STATE FALSE}
DECL E6POS XP808={X 12886.08572,Y -646.4113,Z 3336.02814,A -83.4604,B -12.81532,C -0.94267,S 2,T 35,E1 -10812.08896,E2 0,E3 0,E4 0,E5 0,E6 0}
; DECL LDAT LCPDATP117={VEL 1,ACC 100,APO_DIST 100,APO_FAC 50.0,ORI_TYP #VAR,CIRC_TYP #BASE,JERK_FAC 50.0}
DECL FDAT FP809={TOOL_NO 0,BASE_NO 0,IPO_FRAME #BASE,POINT2[] " ",TQ_STATE FALSE}
DECL E6POS XP809={X 6226.20694,Y -691.76303,Z 3410.82553,A -102.7078,B 7.77597,C 4.76022,S 2,T 35,E1 -4167.06683,E2 0,E3 0,E4 0,E5 0,E6 0}
; DECL LDAT LCPDATP118={VEL 1,ACC 100,APO_DIST 100,APO_FAC 50.0,ORI_TYP #VAR,CIRC_TYP #BASE,JERK_FAC 50.0}
DECL FDAT FP810={TOOL_NO 0,BASE_NO 0,IPO_FRAME #BASE,POINT2[] " ",TQ_STATE FALSE}
DECL E6POS XP810={X 6109.20944,Y -705.3695,Z 3654.40552,A -102.70779,B 7.77597,C 4.76025,S 2,T 35,E1 -4140.9372,E2 0,E3 0,E4 0,E5 0,E6 0}
; DECL LDAT LCPDATP121={VEL 1,ACC 100,APO_DIST 100,APO_FAC 50.0,ORI_TYP #VAR,CIRC_TYP #BASE,JERK_FAC 50.0}
DECL FDAT FP811={TOOL_NO 0,BASE_NO 0,IPO_FRAME #BASE,POINT2[] " ",TQ_STATE FALSE}
DECL E6POS XP811={X 12777.06723,Y -602.17839,Z 3573.69413,A -83.4604,B -12.81532,C -0.94267,S 2,T 35,E1 -10812.08896,E2 0,E3 0,E4 0,E5 0,E6 0}
; DECL LDAT LCPDATP122={VEL 1,ACC 100,APO_DIST 100,APO_FAC 50.0,ORI_TYP #VAR,CIRC_TYP #BASE,JERK_FAC 50.0}
DECL FDAT FP812={TOOL_NO 0,BASE_NO 0,IPO_FRAME #BASE,POINT2[] " ",TQ_STATE FALSE}
DECL E6POS XP812={X 12675.92788,Y -569.18264,Z 3775.2407,A -83.4604,B -12.81532,C -0.94267,S 2,T 35,E1 -10812.08896,E2 0,E3 0,E4 0,E5 0,E6 0}
; DECL LDAT LCPDATP119={VEL 1,ACC 100,APO_DIST 100,APO_FAC 50.0,ORI_TYP #VAR,CIRC_TYP #BASE,JERK_FAC 50.0}
DECL FDAT FP813={TOOL_NO 0,BASE_NO 0,IPO_FRAME #BASE,POINT2[] " ",TQ_STATE FALSE}
DECL E6POS XP813={X 6034.81499,Y -708.12179,Z 3847.76366,A -102.7078,B 7.77596,C 4.76026,S 2,T 35,E1 -4174.36752,E2 0,E3 0,E4 0,E5 0,E6 0}
; DECL LDAT LCPDATP120={VEL 1,ACC 100,APO_DIST 100,APO_FAC 50.0,ORI_TYP #VAR,CIRC_TYP #BASE,JERK_FAC 50.0}
DECL FDAT FP814={TOOL_NO 0,BASE_NO 0,IPO_FRAME #BASE,POINT2[] " ",TQ_STATE FALSE}
DECL E6POS XP814={X 5808.56571,Y -717.10091,Z 4003.7046,A -102.70779,B 7.77596,C 4.76025,S 2,T 35,E1 -4005.10214,E2 0,E3 0,E4 0,E5 0,E6 0}
; DECL LDAT LCPDATP123={VEL 1,ACC 100,APO_DIST 100,APO_FAC 50.0,ORI_TYP #VAR,CIRC_TYP #BASE,JERK_FAC 50.0}
DECL FDAT FP815={TOOL_NO 0,BASE_NO 0,IPO_FRAME #BASE,POINT2[] " ",TQ_STATE FALSE}
DECL E6POS XP815={X 12607.03936,Y -538.48386,Z 3940.5062,A -83.4604,B -12.81532,C -0.94267,S 2,T 35,E1 -10812.08896,E2 0,E3 0,E4 0,E5 0,E6 0}
; DECL LDAT LCPDATP124={VEL 1,ACC 100,APO_DIST 100,APO_FAC 50.0,ORI_TYP #VAR,CIRC_TYP #BASE,JERK_FAC 50.0}
DECL FDAT FP816={TOOL_NO 0,BASE_NO 0,IPO_FRAME #BASE,POINT2[] " ",TQ_STATE FALSE}
DECL E6POS XP816={X 12329.73693,Y -538.48386,Z 3940.5062,A -83.38777,B -15.32829,C -1.2413,S 2,T 35,E1 -10812.08896,E2 0,E3 0,E4 0,E5 0,E6 0}
; DECL LDAT LCPDATP130={VEL 1,ACC 100,APO_DIST 100,APO_FAC 50.0,ORI_TYP #VAR,CIRC_TYP #BASE,JERK_FAC 50.0}
DECL FDAT FP817={TOOL_NO 0,BASE_NO 0,IPO_FRAME #BASE,POINT2[] " ",TQ_STATE FALSE}
DECL E6POS XP817={X 6035.27715,Y -717.10158,Z 4003.70466,A -106.51042,B 6.34838,C 5.00917,S 2,T 35,E1 -4231.81368,E2 0,E3 0,E4 0,E5 0,E6 0}
; DECL LDAT LCPDATP131={VEL 1,ACC 100,APO_DIST 100,APO_FAC 50.0,ORI_TYP #VAR,CIRC_TYP #BASE,JERK_FAC 50.0}
DECL FDAT FP818={TOOL_NO 0,BASE_NO 0,IPO_FRAME #BASE,POINT2[] " ",TQ_STATE FALSE}
DECL E6POS XP818={X 6001.84737,Y -717.10113,Z 4003.70421,A -106.4599,B 4.5615,C 5.54032,S 2,T 35,E1 -4198.38336,E2 0,E3 0,E4 0,E5 0,E6 0}
; DECL LDAT LCPDATP125={VEL 1,ACC 100,APO_DIST 100,APO_FAC 50.0,ORI_TYP #VAR,CIRC_TYP #BASE,JERK_FAC 50.0}
DECL FDAT FP819={TOOL_NO 0,BASE_NO 0,IPO_FRAME #BASE,POINT2[] " ",TQ_STATE FALSE}
DECL E6POS XP819={X 12327.62864,Y -538.48366,Z 3940.50597,A -87.76623,B -17.49847,C -1.50503,S 2,T 35,E1 -10473.34117,E2 0,E3 0,E4 0,E5 0,E6 0}
; DECL LDAT LCPDATP126={VEL 1,ACC 100,APO_DIST 100,APO_FAC 50.0,ORI_TYP #VAR,CIRC_TYP #BASE,JERK_FAC 50.0}
DECL FDAT FP820={TOOL_NO 0,BASE_NO 0,IPO_FRAME #BASE,POINT2[] " ",TQ_STATE FALSE}
DECL E6POS XP820={X 12344.44126,Y -538.48354,Z 3940.50612,A -92.12133,B -19.55447,C -1.59012,S 2,T 35,E1 -10490.15446,E2 0,E3 0,E4 0,E5 0,E6 0}
; DECL LDAT LCPDATP132={VEL 1,ACC 100,APO_DIST 100,APO_FAC 50.0,ORI_TYP #VAR,CIRC_TYP #BASE,JERK_FAC 50.0}
DECL FDAT FP821={TOOL_NO 0,BASE_NO 0,IPO_FRAME #BASE,POINT2[] " ",TQ_STATE FALSE}
DECL E6POS XP821={X 5984.60315,Y -717.10142,Z 4003.7045,A -107.27293,B 2.66443,C 6.10126,S 2,T 35,E1 -4181.13976,E2 0,E3 0,E4 0,E5 0,E6 0}
; DECL LDAT LCPDATP133={VEL 1,ACC 100,APO_DIST 100,APO_FAC 50.0,ORI_TYP #VAR,CIRC_TYP #BASE,JERK_FAC 50.0}
DECL FDAT FP822={TOOL_NO 0,BASE_NO 0,IPO_FRAME #BASE,POINT2[] " ",TQ_STATE FALSE}
DECL E6POS XP822={X 5959.53065,Y -717.10165,Z 4003.70439,A -107.25516,B 0.74219,C 6.69889,S 2,T 35,E1 -4156.06702,E2 0,E3 0,E4 0,E5 0,E6 0}
; DECL LDAT LCPDATP127={VEL 1,ACC 100,APO_DIST 100,APO_FAC 50.0,ORI_TYP #VAR,CIRC_TYP #BASE,JERK_FAC 50.0}
DECL FDAT FP823={TOOL_NO 0,BASE_NO 0,IPO_FRAME #BASE,POINT2[] " ",TQ_STATE FALSE}
DECL E6POS XP823={X 12327.65948,Y -538.48376,Z 3940.50627,A -96.02004,B -21.56802,C -1.50992,S 2,T 35,E1 -10473.37259,E2 0,E3 0,E4 0,E5 0,E6 0}
; DECL LDAT LCPDATP128={VEL 1,ACC 100,APO_DIST 100,APO_FAC 50.0,ORI_TYP #VAR,CIRC_TYP #BASE,JERK_FAC 50.0}
DECL FDAT FP824={TOOL_NO 0,BASE_NO 0,IPO_FRAME #BASE,POINT2[] " ",TQ_STATE FALSE}
DECL E6POS XP824={X 12434.40962,Y -538.48361,Z 3791.38491,A -100.48203,B -23.59142,C -1.27711,S 2,T 35,E1 -10580.12251,E2 0,E3 0,E4 0,E5 0,E6 0}
; DECL LDAT LCPDATP134={VEL 1,ACC 100,APO_DIST 100,APO_FAC 50.0,ORI_TYP #VAR,CIRC_TYP #BASE,JERK_FAC 50.0}
DECL FDAT FP825={TOOL_NO 0,BASE_NO 0,IPO_FRAME #BASE,POINT2[] " ",TQ_STATE FALSE}
DECL E6POS XP825={X 6027.18413,Y -717.10157,Z 4003.70451,A -108.83879,B -1.2655,C 7.3225,S 2,T 35,E1 -4223.72032,E2 0,E3 0,E4 0,E5 0,E6 0}
; DECL LDAT LCPDATP135={VEL 1,ACC 100,APO_DIST 100,APO_FAC 50.0,ORI_TYP #VAR,CIRC_TYP #BASE,JERK_FAC 50.0}
DECL FDAT FP826={TOOL_NO 0,BASE_NO 0,IPO_FRAME #BASE,POINT2[] " ",TQ_STATE FALSE}
DECL E6POS XP826={X 5994.01853,Y -717.10159,Z 4003.70409,A -109.42003,B -3.44272,C 8.06654,S 2,T 35,E1 -4190.55423,E2 0,E3 0,E4 0,E5 0,E6 0}
; DECL LDAT LCPDATP129={VEL 1,ACC 100,APO_DIST 100,APO_FAC 50.0,ORI_TYP #VAR,CIRC_TYP #BASE,JERK_FAC 50.0}
DECL FDAT FP827={TOOL_NO 0,BASE_NO 0,IPO_FRAME #BASE,POINT2[] " ",TQ_STATE FALSE}
DECL E6POS XP827={X 12525.53957,Y -538.48385,Z 3733.39322,A -103.74147,B -24.12805,C -1.24549,S 2,T 35,E1 -10671.25219,E2 0,E3 0,E4 0,E5 0,E6 0}
; DECL LDAT LCPDATP138={VEL 1,ACC 100,APO_DIST 100,APO_FAC 50.0,ORI_TYP #VAR,CIRC_TYP #BASE,JERK_FAC 50.0}
DECL FDAT FP828={TOOL_NO 0,BASE_NO 0,IPO_FRAME #BASE,POINT2[] " ",TQ_STATE FALSE}
DECL E6POS XP828={X 12409.55634,Y -538.48385,Z 3733.39322,A -103.74147,B -24.12805,C -1.24549,S 2,T 35,E1 -10555.26896,E2 0,E3 0,E4 0,E5 0,E6 0}
; DECL LDAT LCPDATP136={VEL 1,ACC 100,APO_DIST 100,APO_FAC 50.0,ORI_TYP #VAR,CIRC_TYP #BASE,JERK_FAC 50.0}
DECL FDAT FP829={TOOL_NO 0,BASE_NO 0,IPO_FRAME #BASE,POINT2[] " ",TQ_STATE FALSE}
DECL E6POS XP829={X 5960.30101,Y -717.10136,Z 4003.70387,A -109.95564,B -5.51238,C 8.79955,S 2,T 35,E1 -4156.83652,E2 0,E3 0,E4 0,E5 0,E6 0}
; DECL LDAT LCPDATP137={VEL 1,ACC 100,APO_DIST 100,APO_FAC 50.0,ORI_TYP #VAR,CIRC_TYP #BASE,JERK_FAC 50.0}
DECL FDAT FP830={TOOL_NO 0,BASE_NO 0,IPO_FRAME #BASE,POINT2[] " ",TQ_STATE FALSE}
DECL E6POS XP830={X 5959.29294,Y -717.10098,Z 4003.70454,A -110.58224,B -7.77816,C 9.62993,S 2,T 35,E1 -4155.82897,E2 0,E3 0,E4 0,E5 0,E6 0}
; DECL LDAT LCPDATP139={VEL 1,ACC 100,APO_DIST 100,APO_FAC 50.0,ORI_TYP #VAR,CIRC_TYP #BASE,JERK_FAC 50.0}
DECL FDAT FP831={TOOL_NO 0,BASE_NO 0,IPO_FRAME #BASE,POINT2[] " ",TQ_STATE FALSE}
DECL E6POS XP831={X 12666.37592,Y -538.48386,Z 3733.39329,A -110.95703,B -23.34196,C -1.63568,S 2,T 35,E1 -10812.08896,E2 0,E3 0,E4 0,E5 0,E6 0}
; DECL LDAT LCPDATP140={VEL 1,ACC 100,APO_DIST 100,APO_FAC 50.0,ORI_TYP #VAR,CIRC_TYP #BASE,JERK_FAC 50.0}
DECL FDAT FP832={TOOL_NO 0,BASE_NO 0,IPO_FRAME #BASE,POINT2[] " ",TQ_STATE FALSE}
DECL E6POS XP832={X 12666.37592,Y -538.48386,Z 3700.25522,A -113.36831,B -23.34196,C -1.63568,S 2,T 35,E1 -10812.08896,E2 0,E3 0,E4 0,E5 0,E6 0}
; DECL LDAT LCPDATP149={VEL 1,ACC 100,APO_DIST 100,APO_FAC 50.0,ORI_TYP #VAR,CIRC_TYP #BASE,JERK_FAC 50.0}
DECL FDAT FP833={TOOL_NO 0,BASE_NO 0,IPO_FRAME #BASE,POINT2[] " ",TQ_STATE FALSE}
DECL E6POS XP833={X 5916.8006,Y -717.10155,Z 4003.70412,A -110.72224,B -10.13455,C 10.52896,S 2,T 35,E1 -4113.33656,E2 0,E3 0,E4 0,E5 0,E6 0}
; DECL LDAT LCPDATP150={VEL 1,ACC 100,APO_DIST 100,APO_FAC 50.0,ORI_TYP #VAR,CIRC_TYP #BASE,JERK_FAC 50.0}
DECL FDAT FP834={TOOL_NO 0,BASE_NO 0,IPO_FRAME #BASE,POINT2[] " ",TQ_STATE FALSE}
DECL E6POS XP834={X 5875.31565,Y -717.1012,Z 4003.70448,A -110.8879,B -12.32973,C 11.37928,S 2,T 35,E1 -4071.85169,E2 0,E3 0,E4 0,E5 0,E6 0}
; DECL LDAT LCPDATP141={VEL 1,ACC 100,APO_DIST 100,APO_FAC 50.0,ORI_TYP #VAR,CIRC_TYP #BASE,JERK_FAC 50.0}
DECL FDAT FP835={TOOL_NO 0,BASE_NO 0,IPO_FRAME #BASE,POINT2[] " ",TQ_STATE FALSE}
DECL E6POS XP835={X 12666.37592,Y -538.48386,Z 3675.40167,A -115.34787,B -23.34196,C -1.63568,S 2,T 35,E1 -10812.08896,E2 0,E3 0,E4 0,E5 0,E6 0}
; DECL LDAT LCPDATP142={VEL 1,ACC 100,APO_DIST 100,APO_FAC 50.0,ORI_TYP #VAR,CIRC_TYP #BASE,JERK_FAC 50.0}
DECL FDAT FP836={TOOL_NO 0,BASE_NO 0,IPO_FRAME #BASE,POINT2[] " ",TQ_STATE FALSE}
DECL E6POS XP836={X 12666.37592,Y -538.48386,Z 3725.10877,A -117.62399,B -22.31862,C -2.21953,S 2,T 35,E1 -10812.08896,E2 0,E3 0,E4 0,E5 0,E6 0}
; DECL LDAT LCPDATP151={VEL 1,ACC 100,APO_DIST 100,APO_FAC 50.0,ORI_TYP #VAR,CIRC_TYP #BASE,JERK_FAC 50.0}
DECL FDAT FP837={TOOL_NO 0,BASE_NO 0,IPO_FRAME #BASE,POINT2[] " ",TQ_STATE FALSE}
DECL E6POS XP837={X 5898.57722,Y -717.10122,Z 4003.70435,A -112.09203,B -14.38754,C 12.19033,S 2,T 35,E1 -4095.11298,E2 0,E3 0,E4 0,E5 0,E6 0}
; DECL LDAT LCPDATP152={VEL 1,ACC 100,APO_DIST 100,APO_FAC 50.0,ORI_TYP #VAR,CIRC_TYP #BASE,JERK_FAC 50.0}
DECL FDAT FP838={TOOL_NO 0,BASE_NO 0,IPO_FRAME #BASE,POINT2[] " ",TQ_STATE FALSE}
DECL E6POS XP838={X 5854.40488,Y -717.10171,Z 4003.70448,A -112.35649,B -16.71303,C 13.17652,S 2,T 35,E1 -4050.94133,E2 0,E3 0,E4 0,E5 0,E6 0}
; DECL LDAT LCPDATP143={VEL 1,ACC 100,APO_DIST 100,APO_FAC 50.0,ORI_TYP #VAR,CIRC_TYP #BASE,JERK_FAC 50.0}
DECL FDAT FP839={TOOL_NO 0,BASE_NO 0,IPO_FRAME #BASE,POINT2[] " ",TQ_STATE FALSE}
DECL E6POS XP839={X 12666.37592,Y -538.48386,Z 3708.53974,A -119.39266,B -22.0406,C -2.38888,S 2,T 35,E1 -10812.08896,E2 0,E3 0,E4 0,E5 0,E6 0}
; DECL LDAT LCPDATP144={VEL 1,ACC 100,APO_DIST 100,APO_FAC 50.0,ORI_TYP #VAR,CIRC_TYP #BASE,JERK_FAC 50.0}
DECL FDAT FP840={TOOL_NO 0,BASE_NO 0,IPO_FRAME #BASE,POINT2[] " ",TQ_STATE FALSE}
DECL E6POS XP840={X 12666.37592,Y -538.48386,Z 3716.82426,A -121.52366,B -21.70131,C -2.61349,S 2,T 35,E1 -10812.08896,E2 0,E3 0,E4 0,E5 0,E6 0}
; DECL LDAT LCPDATP153={VEL 1,ACC 100,APO_DIST 100,APO_FAC 50.0,ORI_TYP #VAR,CIRC_TYP #BASE,JERK_FAC 50.0}
DECL FDAT FP841={TOOL_NO 0,BASE_NO 0,IPO_FRAME #BASE,POINT2[] " ",TQ_STATE FALSE}
DECL E6POS XP841={X 5865.70091,Y -717.10124,Z 4003.70383,A -113.62634,B -18.80667,C 14.08679,S 2,T 35,E1 -4062.23613,E2 0,E3 0,E4 0,E5 0,E6 0}
; DECL LDAT LCPDATP154={VEL 1,ACC 100,APO_DIST 100,APO_FAC 50.0,ORI_TYP #VAR,CIRC_TYP #BASE,JERK_FAC 50.0}
DECL FDAT FP842={TOOL_NO 0,BASE_NO 0,IPO_FRAME #BASE,POINT2[] " ",TQ_STATE FALSE}
DECL E6POS XP842={X 5786.97193,Y -717.10138,Z 4003.70442,A -113.90846,B -20.59534,C 14.92344,S 2,T 35,E1 -3983.50839,E2 0,E3 0,E4 0,E5 0,E6 0}
; DECL LDAT LCPDATP145={VEL 1,ACC 100,APO_DIST 100,APO_FAC 50.0,ORI_TYP #VAR,CIRC_TYP #BASE,JERK_FAC 50.0}
DECL FDAT FP843={TOOL_NO 0,BASE_NO 0,IPO_FRAME #BASE,POINT2[] " ",TQ_STATE FALSE}
DECL E6POS XP843={X 12666.37592,Y -538.48386,Z 3691.97071,A -122.58569,B -21.70131,C -2.61349,S 2,T 35,E1 -10812.08896,E2 0,E3 0,E4 0,E5 0,E6 0}
; DECL LDAT LCPDATP146={VEL 1,ACC 100,APO_DIST 100,APO_FAC 50.0,ORI_TYP #VAR,CIRC_TYP #BASE,JERK_FAC 50.0}
DECL FDAT FP844={TOOL_NO 0,BASE_NO 0,IPO_FRAME #BASE,POINT2[] " ",TQ_STATE FALSE}
DECL E6POS XP844={X 12666.37592,Y -538.48386,Z 3741.67781,A -124.88801,B -20.60151,C -3.44033,S 2,T 35,E1 -10812.08896,E2 0,E3 0,E4 0,E5 0,E6 0}
; DECL LDAT LCPDATP155={VEL 1,ACC 100,APO_DIST 100,APO_FAC 50.0,ORI_TYP #VAR,CIRC_TYP #BASE,JERK_FAC 50.0}
DECL FDAT FP845={TOOL_NO 0,BASE_NO 0,IPO_FRAME #BASE,POINT2[] " ",TQ_STATE FALSE}
DECL E6POS XP845={X 5766.06143,Y -717.10078,Z 4003.7047,A -114.88478,B -21.82725,C 15.51221,S 2,T 35,E1 -3962.59803,E2 0,E3 0,E4 0,E5 0,E6 0}
; DECL LDAT LCPDATP156={VEL 1,ACC 100,APO_DIST 100,APO_FAC 50.0,ORI_TYP #VAR,CIRC_TYP #BASE,JERK_FAC 50.0}
DECL FDAT FP846={TOOL_NO 0,BASE_NO 0,IPO_FRAME #BASE,POINT2[] " ",TQ_STATE FALSE}
DECL E6POS XP846={X 5671.46198,Y -717.1018,Z 4003.704,A -116.65787,B -23.21109,C 16.21129,S 2,T 35,E1 -3867.99764,E2 0,E3 0,E4 0,E5 0,E6 0}
; DECL LDAT LCPDATP147={VEL 1,ACC 100,APO_DIST 100,APO_FAC 50.0,ORI_TYP #VAR,CIRC_TYP #BASE,JERK_FAC 50.0}
DECL FDAT FP847={TOOL_NO 0,BASE_NO 0,IPO_FRAME #BASE,POINT2[] " ",TQ_STATE FALSE}
DECL E6POS XP847={X 12666.37592,Y -538.48386,Z 3708.53974,A -127.07895,B -20.60151,C -3.44033,S 2,T 35,E1 -10812.08896,E2 0,E3 0,E4 0,E5 0,E6 0}

ENDDAT
